C09152=1181.031,74.990,-49.573,-179.182,6.039,148.840
C09153=1181.026,75.239,-49.589,-179.180,6.040,148.840
C09154=1181.021,75.489,-49.607,-179.177,6.041,148.839
C09155=1181.017,75.738,-49.624,-179.175,6.042,148.839
C09156=1181.011,75.987,-49.641,-179.171,6.043,148.838
C09157=1181.006,76.236,-49.659,-179.169,6.044,148.838
C09158=1181.001,76.486,-49.676,-179.167,6.045,148.837
C09159=1180.996,76.736,-49.693,-179.164,6.047,148.837
C09160=1180.992,76.985,-49.710,-179.161,6.047,148.836
C09161=1180.987,77.234,-49.727,-179.159,6.049,148.836
C09162=1180.981,77.483,-49.744,-179.156,6.049,148.835
C09163=1180.977,77.732,-49.762,-179.153,6.051,148.835
C09164=1180.972,77.982,-49.779,-179.151,6.052,148.834
C09165=1180.966,78.232,-49.796,-179.149,6.052,148.834
C09166=1180.962,78.481,-49.814,-179.145,6.054,148.833
C09167=1180.957,78.731,-49.831,-179.143,6.055,148.832
C09168=1180.952,78.980,-49.849,-179.140,6.056,148.832
C09169=1180.948,79.229,-49.866,-179.138,6.057,148.831
C09170=1180.942,79.478,-49.882,-179.135,6.057,148.831
C09171=1180.937,79.727,-49.900,-179.132,6.059,148.830
C09172=1180.932,79.977,-49.917,-179.130,6.060,148.830
C09173=1180.927,80.245,-49.937,-179.127,6.061,148.829
C09174=1180.922,80.514,-49.955,-179.124,6.063,148.829
C09175=1180.916,80.782,-49.974,-179.121,6.063,148.828
C09176=1180.912,81.050,-49.992,-179.119,6.065,148.828
C09177=1180.906,81.300,-50.010,-179.116,6.066,148.827
C09178=1180.901,81.549,-50.028,-179.113,6.067,148.826
C09179=1180.896,81.799,-50.045,-179.111,6.068,148.826
C09180=1180.892,82.048,-50.062,-179.108,6.070,148.825
C09181=1180.887,82.298,-50.080,-179.105,6.070,148.825
C09182=1180.882,82.547,-50.097,-179.103,6.071,148.824
C09183=1180.877,82.796,-50.114,-179.100,6.072,148.824
C09184=1180.873,83.045,-50.132,-179.098,6.073,148.823
C09185=1180.868,83.295,-50.150,-179.095,6.075,148.823
C09186=1180.862,83.544,-50.167,-179.092,6.075,148.822
C09187=1180.858,83.794,-50.185,-179.090,6.077,148.822
C09188=1180.853,84.043,-50.202,-179.087,6.078,148.821
C09189=1180.848,84.292,-50.220,-179.084,6.079,148.821
C09190=1180.843,84.541,-50.238,-179.082,6.080,148.820
C09191=1180.837,84.790,-50.255,-179.079,6.082,148.820
C09192=1180.832,85.040,-50.273,-179.076,6.082,148.819
C09193=1180.828,85.289,-50.290,-179.074,6.083,148.818
C09194=1180.823,85.538,-50.308,-179.071,6.084,148.818
C09195=1180.818,85.787,-50.325,-179.069,6.085,148.817
C09196=1180.813,86.037,-50.343,-179.066,6.087,148.817
C09197=1180.808,86.286,-50.361,-179.064,6.088,148.816
C09198=1180.804,86.536,-50.379,-179.060,6.089,148.816
C09199=1180.800,86.785,-50.396,-179.058,6.090,148.815
C09200=1180.794,87.035,-50.414,-179.055,6.092,148.815
C09201=1180.789,87.284,-50.432,-179.053,6.092,148.814
C09202=1180.785,87.533,-50.450,-179.050,6.094,148.814
C09203=1180.780,87.783,-50.468,-179.048,6.094,148.813
C09204=1180.774,88.032,-50.485,-179.045,6.096,148.813
C09205=1180.769,88.282,-50.503,-179.042,6.097,148.812
C09206=1180.765,88.531,-50.521,-179.039,6.098,148.812
C09207=1180.760,88.780,-50.539,-179.037,6.099,148.811
C09208=1180.755,89.029,-50.557,-179.034,6.101,148.811
C09209=1180.750,89.279,-50.574,-179.031,6.101,148.810
C09210=1180.745,89.528,-50.592,-179.029,6.103,148.810
C09211=1180.740,89.777,-50.609,-179.027,6.104,148.809
C09212=1180.736,90.026,-50.627,-179.023,6.105,148.808
C09213=1180.731,90.275,-50.645,-179.021,6.106,148.808
C09214=1180.726,90.524,-50.663,-179.018,6.107,148.807
C09215=1180.720,90.774,-50.681,-179.016,6.108,148.807
C09216=1180.716,91.024,-50.699,-179.013,6.110,148.806
C09217=1180.711,91.273,-50.717,-179.011,6.111,148.806
C09218=1180.706,91.522,-50.735,-179.008,6.112,148.805
C09219=1180.701,91.772,-50.753,-179.005,6.113,148.805
C09220=1180.697,92.021,-50.771,-179.003,6.115,148.804
C09221=1180.692,92.270,-50.789,-179.000,6.115,148.804
C09222=1180.687,92.519,-50.807,-178.997,6.117,148.803
C09223=1180.682,92.768,-50.825,-178.995,6.117,148.803
C09224=1180.677,93.017,-50.843,-178.992,6.119,148.802
C09225=1180.673,93.267,-50.861,-178.990,6.120,148.802
C09226=1180.668,93.517,-50.879,-178.987,6.121,148.801
C09227=1180.663,93.766,-50.897,-178.984,6.122,148.801
C09228=1180.658,94.015,-50.915,-178.981,6.124,148.800
C09229=1180.652,94.264,-50.934,-178.979,6.125,148.800
C09230=1180.647,94.514,-50.952,-178.976,6.126,148.799
C09231=1180.642,94.763,-50.970,-178.974,6.127,148.799
C09232=1180.638,95.013,-50.988,-178.971,6.129,148.798
C09233=1180.633,95.262,-51.006,-178.968,6.129,148.798
C09234=1180.628,95.511,-51.024,-178.966,6.131,148.797
C09235=1180.623,95.760,-51.042,-178.963,6.131,148.797
C09236=1180.618,96.009,-51.060,-178.960,6.133,148.796
C09237=1180.613,96.258,-51.078,-178.958,6.134,148.795
C09238=1180.609,96.508,-51.096,-178.955,6.135,148.795
C09239=1180.604,96.758,-51.115,-178.952,6.137,148.795
C09240=1180.599,97.007,-51.133,-178.950,6.138,148.794
C09241=1180.594,97.256,-51.151,-178.947,6.139,148.794
C09242=1180.589,97.505,-51.169,-178.944,6.140,148.793
C09243=1180.585,97.755,-51.188,-178.942,6.142,148.793
C09244=1180.580,98.004,-51.206,-178.939,6.143,148.792
C09245=1180.574,98.253,-51.224,-178.936,6.144,148.791
C09246=1180.569,98.502,-51.242,-178.934,6.145,148.791
C09247=1180.565,98.752,-51.261,-178.931,6.146,148.790
C09248=1180.560,99.002,-51.279,-178.929,6.147,148.790
C09249=1180.555,99.250,-51.297,-178.926,6.149,148.790
C09250=1180.551,99.499,-51.315,-178.923,6.150,148.789
C09251=1180.545,99.749,-51.334,-178.921,6.151,148.789
C09252=1180.541,99.999,-51.352,-178.918,6.152,148.788
C09253=1180.536,100.247,-51.371,-178.915,6.153,148.787
C09254=1180.531,100.496,-51.389,-178.913,6.155,148.787
C09255=1180.526,100.747,-51.408,-178.910,6.156,148.786
C09256=1180.521,100.996,-51.426,-178.907,6.157,148.786
C09257=1180.517,101.244,-51.445,-178.905,6.158,148.786
C09258=1180.512,101.493,-51.463,-178.902,6.160,148.785
C09259=1180.507,101.744,-51.482,-178.899,6.161,148.785
C09260=1180.502,101.992,-51.500,-178.897,6.162,148.784
C09261=1180.497,102.241,-51.518,-178.894,6.164,148.784
C09262=1180.492,102.491,-51.536,-178.892,6.165,148.783
C09263=1180.487,102.740,-51.556,-178.889,6.166,148.782
C09264=1180.482,102.989,-51.574,-178.887,6.167,148.782
C09265=1180.478,103.238,-51.592,-178.883,6.168,148.781
C09266=1180.473,103.488,-51.611,-178.881,6.170,148.781
C09267=1180.468,103.737,-51.629,-178.879,6.171,148.781
C09268=1180.463,103.986,-51.647,-178.875,6.172,148.780
C09269=1180.458,104.236,-51.667,-178.873,6.173,148.780
C09270=1180.453,104.485,-51.685,-178.870,6.175,148.779
C09271=1180.449,104.734,-51.704,-178.867,6.176,148.778
C09272=1180.444,104.984,-51.723,-178.865,6.177,148.778
C09273=1180.439,105.233,-51.741,-178.862,6.179,148.778
C09274=1180.433,105.482,-51.760,-178.860,6.179,148.777
C09275=1180.429,105.732,-51.778,-178.857,6.181,148.777
C09276=1180.425,105.980,-51.797,-178.854,6.183,148.776
C09277=1180.419,106.249,-51.817,-178.852,6.183,148.776
C09278=1180.415,106.517,-51.837,-178.849,6.185,148.775
C09279=1180.409,106.786,-51.858,-178.846,6.187,148.775
C09280=1180.403,107.054,-51.878,-178.843,6.188,148.774
C09281=1180.399,107.304,-51.897,-178.841,6.189,148.773
C09282=1180.394,107.553,-51.915,-178.838,6.191,148.773
C09283=1180.389,107.802,-51.934,-178.835,6.192,148.772
C09284=1180.385,108.051,-51.953,-178.833,6.193,148.772
C09285=1180.379,108.300,-51.971,-178.830,6.195,148.772
C09286=1180.375,108.550,-51.991,-178.827,6.195,148.771
C09287=1180.369,108.799,-52.009,-178.824,6.197,148.771
C09288=1180.365,109.048,-52.028,-178.821,6.198,148.770
C09289=1180.360,109.298,-52.047,-178.819,6.199,148.770
C09290=1180.355,109.546,-52.065,-178.816,6.201,148.769
C09291=1180.350,109.796,-52.085,-178.814,6.202,148.768
C09292=1180.345,110.045,-52.103,-178.811,6.203,148.768
C09293=1180.341,110.295,-52.123,-178.808,6.205,148.768
C09294=1180.336,110.543,-52.141,-178.806,6.206,148.767
C09295=1180.330,110.793,-52.160,-178.803,6.207,148.767
C09296=1180.326,111.042,-52.179,-178.800,6.209,148.766
C09297=1180.321,111.291,-52.198,-178.798,6.210,148.766
C09298=1180.317,111.541,-52.217,-178.795,6.211,148.765
C09299=1180.311,111.790,-52.236,-178.792,6.213,148.765
C09300=1180.307,112.039,-52.255,-178.790,6.214,148.764
C09301=1180.302,112.288,-52.274,-178.787,6.215,148.764
C09302=1180.298,112.538,-52.293,-178.785,6.216,148.763
C09303=1180.292,112.787,-52.312,-178.782,6.218,148.763
C09304=1180.288,113.036,-52.332,-178.779,6.219,148.762
C09305=1180.283,113.285,-52.350,-178.777,6.220,148.762
C09306=1180.278,113.535,-52.369,-178.774,6.222,148.761
C09307=1180.273,113.783,-52.388,-178.771,6.223,148.761
C09308=1180.269,114.033,-52.408,-178.769,6.224,148.760
C09309=1180.263,114.282,-52.427,-178.766,6.226,148.760
C09310=1180.259,114.532,-52.445,-178.763,6.227,148.759
C09311=1180.254,114.781,-52.465,-178.761,6.228,148.759
C09312=1180.249,115.030,-52.484,-178.758,6.230,148.759
C09313=1180.244,115.279,-52.503,-178.755,6.231,148.758
C09314=1180.240,115.528,-52.523,-178.753,6.232,148.758
C09315=1180.234,115.777,-52.542,-178.750,6.234,148.757
C09316=1180.230,116.026,-52.561,-178.747,6.235,148.757
C09317=1180.225,116.276,-52.579,-178.745,6.236,148.756
C09318=1180.220,116.525,-52.599,-178.742,6.238,148.756
C09319=1180.215,116.774,-52.618,-178.739,6.240,148.755
C09320=1180.210,117.024,-52.637,-178.737,6.240,148.755
C09321=1180.205,117.272,-52.657,-178.734,6.242,148.754
C09322=1180.201,117.522,-52.676,-178.731,6.244,148.754
C09323=1180.196,117.771,-52.696,-178.729,6.244,148.753
C09324=1180.191,118.020,-52.715,-178.726,6.246,148.753
C09325=1180.186,118.270,-52.734,-178.723,6.248,148.752
C09326=1180.182,118.518,-52.753,-178.721,6.249,148.752
C09327=1180.177,118.768,-52.773,-178.718,6.250,148.751
C09328=1180.172,119.017,-52.792,-178.715,6.252,148.751
C09329=1180.167,119.266,-52.812,-178.713,6.253,148.751
C09330=1180.163,119.516,-52.831,-178.710,6.254,148.750
C09331=1180.157,119.764,-52.850,-178.707,6.256,148.750
C09332=1180.153,120.014,-52.870,-178.705,6.257,148.749
C09333=1180.147,120.263,-52.889,-178.702,6.258,148.749
C09334=1180.143,120.512,-52.908,-178.699,6.260,148.748
C09335=1180.139,120.762,-52.928,-178.697,6.261,148.748
C09336=1180.133,121.011,-52.947,-178.694,6.263,148.747
C09337=1180.129,121.260,-52.967,-178.691,6.264,148.747
C09338=1180.124,121.510,-52.986,-178.689,6.266,148.746
C09339=1180.119,121.758,-53.005,-178.686,6.267,148.746
C09340=1180.115,122.007,-53.025,-178.683,6.268,148.745
C09341=1180.110,122.257,-53.045,-178.681,6.270,148.745
C09342=1180.105,122.506,-53.064,-178.678,6.271,148.744
C09343=1180.100,122.755,-53.084,-178.676,6.273,148.744
C09344=1180.095,123.005,-53.104,-178.673,6.274,148.743
C09345=1180.090,123.254,-53.123,-178.670,6.276,148.743
C09346=1180.086,123.502,-53.143,-178.668,6.277,148.743
C09347=1180.081,123.752,-53.162,-178.665,6.278,148.742
C09348=1180.076,124.001,-53.182,-178.662,6.280,148.742
C09349=1180.071,124.250,-53.201,-178.660,6.281,148.741
C09350=1180.067,124.500,-53.221,-178.657,6.282,148.741
C09351=1180.062,124.748,-53.241,-178.654,6.284,148.740
C09352=1180.057,124.998,-53.261,-178.651,6.286,148.740
C09353=1180.052,125.247,-53.280,-178.649,6.287,148.739
C09354=1180.047,125.496,-53.300,-178.646,6.288,148.739
C09355=1180.042,125.745,-53.320,-178.644,6.290,148.739
C09356=1180.038,125.995,-53.340,-178.641,6.291,148.738
C09357=1180.034,126.244,-53.359,-178.638,6.292,148.738
C09358=1180.028,126.492,-53.379,-178.636,6.294,148.737
C09359=1180.024,126.742,-53.398,-178.633,6.296,148.737
C09360=1180.019,126.991,-53.418,-178.630,6.296,148.736
C09361=1180.014,127.239,-53.438,-178.628,6.298,148.736
C09362=1180.009,127.489,-53.458,-178.625,6.300,148.735
C09363=1180.004,127.739,-53.477,-178.622,6.302,148.735
C09364=1180.000,127.988,-53.498,-178.620,6.302,148.734
C09365=1179.995,128.237,-53.517,-178.617,6.304,148.734
C09366=1179.990,128.486,-53.537,-178.614,6.306,148.734
C09367=1179.986,128.735,-53.557,-178.611,6.307,148.733
C09368=1179.981,128.985,-53.577,-178.609,6.308,148.733
C09369=1179.976,129.233,-53.597,-178.606,6.310,148.732
C09370=1179.971,129.482,-53.616,-178.603,6.311,148.732
C09371=1179.967,129.731,-53.637,-178.601,6.313,148.731
C09372=1179.961,129.981,-53.657,-178.599,6.314,148.731
C09373=1179.956,130.231,-53.677,-178.595,6.316,148.730
C09374=1179.952,130.480,-53.697,-178.593,6.317,148.730
C09375=1179.947,130.729,-53.716,-178.590,6.319,148.730
C09376=1179.942,130.977,-53.737,-178.588,6.320,148.729
C09377=1179.937,131.227,-53.756,-178.585,6.321,148.729
C09378=1179.933,131.476,-53.777,-178.582,6.323,148.728
C09379=1179.928,131.726,-53.796,-178.579,6.325,148.728
C09380=1179.923,131.974,-53.816,-178.577,6.326,148.727
C09381=1179.917,132.243,-53.838,-178.574,6.327,148.727
C09382=1179.913,132.511,-53.860,-178.571,6.329,148.726
C09383=1179.907,132.780,-53.882,-178.569,6.331,148.726
C09384=1179.902,133.048,-53.903,-178.565,6.332,148.725
C09385=1179.898,133.297,-53.923,-178.563,6.334,148.725
C09386=1179.893,133.547,-53.944,-178.560,6.336,148.725
C09387=1179.888,133.796,-53.964,-178.557,6.337,148.724
C09388=1179.884,134.045,-53.984,-178.554,6.339,148.724
C09389=1179.879,134.295,-54.004,-178.552,6.340,148.723
C09390=1179.874,134.544,-54.024,-178.549,6.341,148.723
C09391=1179.869,134.793,-54.045,-178.547,6.343,148.722
C09392=1179.864,135.042,-54.064,-178.544,6.345,148.722
C09393=1179.859,135.291,-54.085,-178.541,6.346,148.721
C09394=1179.855,135.540,-54.105,-178.539,6.347,148.721
C09395=1179.851,135.789,-54.125,-178.536,6.349,148.721
C09396=1179.845,136.039,-54.146,-178.533,6.351,148.720
C09397=1179.841,136.287,-54.166,-178.531,6.352,148.720
C09398=1179.836,136.536,-54.186,-178.528,6.354,148.719
C09399=1179.831,136.786,-54.206,-178.525,6.355,148.719
C09400=1179.826,137.035,-54.227,-178.523,6.357,148.718
C09401=1179.822,137.284,-54.247,-178.520,6.358,148.718
C09402=1179.817,137.532,-54.267,-178.517,6.360,148.718
C09403=1179.812,137.782,-54.287,-178.514,6.362,148.717
C09404=1179.807,138.031,-54.308,-178.512,6.362,148.717
C09405=1179.802,138.280,-54.328,-178.509,6.364,148.716
C09406=1179.798,138.529,-54.349,-178.506,6.366,148.716
C09407=1179.793,138.778,-54.370,-178.504,6.368,148.715
C09408=1179.788,139.027,-54.390,-178.501,6.369,148.715
C09409=1179.784,139.277,-54.410,-178.499,6.370,148.715
C09410=1179.778,139.526,-54.431,-178.496,6.372,148.714
C09411=1179.774,139.775,-54.451,-178.493,6.373,148.714
C09412=1179.770,140.024,-54.471,-178.490,6.375,148.713
C09413=1179.764,140.273,-54.492,-178.488,6.377,148.713
C09414=1179.760,140.522,-54.513,-178.485,6.379,148.712
C09415=1179.756,140.771,-54.533,-178.483,6.380,148.712
C09416=1179.750,141.021,-54.554,-178.480,6.381,148.711
C09417=1179.746,141.269,-54.575,-178.477,6.383,148.711
C09418=1179.740,141.519,-54.595,-178.474,6.385,148.711
C09419=1179.736,141.768,-54.615,-178.472,6.386,148.710
C09420=1179.732,142.017,-54.635,-178.469,6.388,148.710
C09421=1179.726,142.267,-54.656,-178.467,6.389,148.710
C09422=1179.722,142.515,-54.677,-178.464,6.391,148.709
C09423=1179.717,142.765,-54.698,-178.461,6.392,148.709
C09424=1179.712,143.014,-54.718,-178.458,6.394,148.708
C09425=1179.708,143.263,-54.739,-178.456,6.396,148.708
C09426=1179.703,143.512,-54.760,-178.453,6.397,148.707
C09427=1179.698,143.761,-54.780,-178.450,6.399,148.707
C09428=1179.693,144.010,-54.801,-178.448,6.400,148.707
C09429=1179.689,144.258,-54.822,-178.445,6.402,148.706
C09430=1179.684,144.508,-54.843,-178.442,6.403,148.706
C09431=1179.679,144.757,-54.863,-178.440,6.405,148.705
C09432=1179.675,145.007,-54.885,-178.437,6.407,148.705
C09433=1179.670,145.256,-54.905,-178.434,6.409,148.704
C09434=1179.665,145.505,-54.926,-178.431,6.410,148.704
C09435=1179.661,145.754,-54.946,-178.429,6.411,148.704
C09436=1179.656,146.003,-54.967,-178.427,6.413,148.703
C09437=1179.651,146.252,-54.988,-178.424,6.415,148.703
C09438=1179.646,146.501,-55.009,-178.421,6.416,148.702
C09439=1179.642,146.750,-55.030,-178.418,6.418,148.702
C09440=1179.637,146.999,-55.051,-178.415,6.420,148.702
C09441=1179.632,147.248,-55.071,-178.413,6.421,148.701
C09442=1179.627,147.497,-55.092,-178.411,6.422,148.701
C09443=1179.622,147.747,-55.113,-178.408,6.424,148.700
C09444=1179.618,147.995,-55.134,-178.405,6.426,148.700
C09445=1179.613,148.245,-55.155,-178.402,6.428,148.700
C09446=1179.609,148.494,-55.176,-178.399,6.429,148.699
C09447=1179.604,148.743,-55.197,-178.397,6.431,148.699
C09448=1179.599,148.991,-55.218,-178.394,6.433,148.698
C09449=1179.594,149.240,-55.239,-178.391,6.434,148.698
C09450=1179.589,149.490,-55.260,-178.389,6.436,148.698
C09451=1179.585,149.739,-55.281,-178.386,6.437,148.697
C09452=1179.580,149.988,-55.302,-178.384,6.439,148.697
C09453=1179.575,150.237,-55.323,-178.381,6.441,148.696
C09454=1179.571,150.486,-55.344,-178.378,6.442,148.696
C09455=1179.566,150.735,-55.365,-178.376,6.444,148.696
C09456=1179.561,150.984,-55.386,-178.373,6.446,148.695
C09457=1179.557,151.234,-55.407,-178.370,6.447,148.695
C09458=1179.552,151.482,-55.429,-178.367,6.449,148.694
C09459=1179.547,151.732,-55.450,-178.364,6.451,148.694
C09460=1179.543,151.980,-55.471,-178.362,6.453,148.693
C09461=1179.538,152.229,-55.492,-178.360,6.453,148.693
C09462=1179.533,152.479,-55.513,-178.357,6.455,148.693
C09463=1179.528,152.728,-55.535,-178.354,6.457,148.692
C09464=1179.524,152.977,-55.555,-178.352,6.459,148.692
C09465=1179.519,153.225,-55.577,-178.349,6.461,148.692
C09466=1179.514,153.475,-55.598,-178.346,6.462,148.691
C09467=1179.509,153.724,-55.620,-178.344,6.464,148.691
C09468=1179.505,153.973,-55.640,-178.341,6.466,148.690
C09469=1179.500,154.222,-55.662,-178.338,6.467,148.690
C09470=1179.495,154.471,-55.683,-178.335,6.469,148.689
C09471=1179.491,154.720,-55.705,-178.332,6.471,148.689
C09472=1179.486,154.969,-55.725,-178.330,6.473,148.689
C09473=1179.481,155.218,-55.747,-178.327,6.474,148.688
C09474=1179.476,155.467,-55.768,-178.325,6.475,148.688
C09475=1179.472,155.716,-55.790,-178.322,6.477,148.688
C09476=1179.467,155.966,-55.811,-178.319,6.479,148.687
C09477=1179.462,156.214,-55.832,-178.317,6.480,148.687
C09478=1179.457,156.463,-55.853,-178.314,6.482,148.686
C09479=1179.453,156.713,-55.875,-178.311,6.484,148.686
C09480=1179.448,156.961,-55.897,-178.309,6.486,148.686
C09481=1179.443,157.210,-55.918,-178.306,6.488,148.685
C09482=1179.439,157.460,-55.940,-178.303,6.489,148.685
C09483=1179.434,157.708,-55.961,-178.301,6.491,148.685
C09484=1179.429,157.958,-55.982,-178.298,6.493,148.684
C09485=1179.424,158.227,-56.005,-178.295,6.494,148.684
C09486=1179.420,158.495,-56.028,-178.292,6.496,148.683
C09487=1179.414,158.764,-56.052,-178.289,6.498,148.683
C09488=1179.409,159.034,-56.075,-178.286,6.500,148.683
C09489=1179.404,159.282,-56.096,-178.283,6.502,148.682
C09490=1179.400,159.532,-56.118,-178.281,6.504,148.682
C09491=1179.395,159.781,-56.139,-178.278,6.506,148.681
C09492=1179.390,160.029,-56.161,-178.276,6.507,148.681
C09493=1179.386,160.279,-56.183,-178.273,6.508,148.681
C09494=1179.381,160.527,-56.205,-178.271,6.510,148.680
C09495=1179.376,160.776,-56.226,-178.268,6.512,148.680
C09496=1179.372,161.026,-56.248,-178.265,6.514,148.680
C09497=1179.367,161.275,-56.269,-178.263,6.515,148.679
C09498=1179.362,161.523,-56.291,-178.260,6.517,148.679
C09499=1179.358,161.773,-56.313,-178.257,6.519,148.678
C09500=1179.353,162.021,-56.335,-178.254,6.520,148.678
C09501=1179.348,162.271,-56.356,-178.251,6.522,148.677
C09502=1179.343,162.520,-56.378,-178.249,6.524,148.677
C09503=1179.338,162.769,-56.400,-178.246,6.526,148.677
C09504=1179.334,163.018,-56.422,-178.243,6.527,148.676
C09505=1179.329,163.266,-56.443,-178.241,6.529,148.676
C09506=1179.325,163.516,-56.465,-178.238,6.531,148.676
C09507=1179.320,163.764,-56.487,-178.235,6.533,148.675
C09508=1179.316,164.014,-56.509,-178.233,6.535,148.675
C09509=1179.311,164.262,-56.531,-178.230,6.536,148.674
C09510=1179.306,164.512,-56.552,-178.227,6.538,148.674
C09511=1179.302,164.761,-56.574,-178.224,6.540,148.674
C09512=1179.297,165.010,-56.595,-178.222,6.542,148.673
C09513=1179.292,165.259,-56.617,-178.219,6.543,148.673
C09514=1179.287,165.508,-56.640,-178.216,6.545,148.673
C09515=1179.282,165.757,-56.662,-178.214,6.547,148.672
C09516=1179.278,166.006,-56.683,-178.211,6.549,148.672
C09517=1179.273,166.255,-56.706,-178.208,6.550,148.671
C09518=1179.268,166.504,-56.727,-178.206,6.552,148.671
C09519=1179.264,166.753,-56.749,-178.203,6.554,148.671
C09520=1179.260,167.001,-56.772,-178.201,6.556,148.671
C09521=1179.255,167.250,-56.793,-178.198,6.558,148.670
C09522=1179.250,167.500,-56.816,-178.195,6.560,148.670
C09523=1179.245,167.748,-56.838,-178.193,6.561,148.670
C09524=1179.241,167.998,-56.860,-178.190,6.563,148.669
C09525=1179.236,168.246,-56.881,-178.187,6.565,148.669
C09526=1179.232,168.496,-56.903,-178.185,6.567,148.668
C09527=1179.226,168.745,-56.926,-178.182,6.568,148.668
C09528=1179.222,168.994,-56.948,-178.179,6.570,148.668
C09529=1179.217,169.242,-56.969,-178.177,6.572,148.667
C09530=1179.213,169.491,-56.992,-178.174,6.574,148.667
C09531=1179.209,169.741,-57.014,-178.171,6.576,148.667
C09532=1179.203,169.990,-57.037,-178.169,6.577,148.666
C09533=1179.199,170.239,-57.059,-178.166,6.579,148.666
C09534=1179.194,170.487,-57.080,-178.163,6.582,148.665
C09535=1179.190,170.736,-57.103,-178.160,6.583,148.665
C09536=1179.184,170.985,-57.125,-178.157,6.585,148.665
C09537=1179.180,171.235,-57.147,-178.155,6.587,148.664
C09538=1179.175,171.483,-57.169,-178.152,6.589,148.664
C09539=1179.170,171.732,-57.192,-178.149,6.591,148.664
C09540=1179.166,171.981,-57.214,-178.147,6.592,148.663
C09541=1179.161,172.230,-57.236,-178.144,6.594,148.663
C09542=1179.157,172.480,-57.258,-178.141,6.596,148.663
C09543=1179.152,172.728,-57.281,-178.139,6.598,148.662
C09544=1179.147,172.977,-57.303,-178.136,6.599,148.662
C09545=1179.143,173.226,-57.325,-178.134,6.602,148.662
C09546=1179.138,173.475,-57.348,-178.131,6.603,148.661
C09547=1179.134,173.724,-57.370,-178.128,6.605,148.661
C09548=1179.129,173.973,-57.392,-178.126,6.607,148.661
C09549=1179.124,174.222,-57.415,-178.123,6.609,148.660
C09550=1179.119,174.470,-57.437,-178.120,6.610,148.660
C09551=1179.114,174.720,-57.460,-178.118,6.612,148.660
C09552=1179.110,174.969,-57.482,-178.115,6.614,148.659
C09553=1179.105,175.218,-57.504,-178.112,6.617,148.659
C09554=1179.101,175.467,-57.527,-178.109,6.618,148.658
C09555=1179.096,175.716,-57.550,-178.106,6.620,148.658
C09556=1179.091,175.964,-57.573,-178.104,6.622,148.658
C09557=1179.087,176.214,-57.595,-178.101,6.624,148.657
C09558=1179.083,176.462,-57.617,-178.099,6.626,148.657
C09559=1179.077,176.711,-57.640,-178.096,6.628,148.657
C09560=1179.073,176.960,-57.662,-178.093,6.629,148.656
C09561=1179.068,177.210,-57.685,-178.091,6.631,148.656
C09562=1179.064,177.458,-57.707,-178.088,6.633,148.656
C09563=1179.059,177.707,-57.730,-178.085,6.635,148.655
C09564=1179.055,177.956,-57.753,-178.083,6.636,148.655
C09565=1179.049,178.205,-57.775,-178.080,6.638,148.655
C09566=1179.045,178.454,-57.798,-178.077,6.641,148.654
C09567=1179.040,178.703,-57.821,-178.074,6.643,148.654
C09568=1179.036,178.951,-57.843,-178.071,6.644,148.654
C09569=1179.031,179.200,-57.866,-178.069,6.646,148.653
C09570=1179.027,179.450,-57.888,-178.067,6.648,148.653
C09571=1179.022,179.699,-57.912,-178.064,6.650,148.653
C09572=1179.017,179.947,-57.934,-178.061,6.652,148.652
C09573=1179.012,180.196,-57.957,-178.059,6.654,148.652
C09574=1179.008,180.445,-57.979,-178.056,6.655,148.652
C09575=1179.003,180.695,-58.002,-178.053,6.657,148.651
C09576=1178.999,180.943,-58.025,-178.050,6.660,148.651
C09577=1178.994,181.192,-58.048,-178.047,6.662,148.651
C09578=1178.989,181.441,-58.071,-178.045,6.664,148.651
C09579=1178.985,181.690,-58.093,-178.042,6.665,148.650
C09580=1178.980,181.939,-58.116,-178.040,6.667,148.650
C09581=1178.976,182.187,-58.139,-178.037,6.669,148.649
C09582=1178.971,182.437,-58.162,-178.034,6.671,148.649
C09583=1178.966,182.686,-58.185,-178.032,6.673,148.649
C09584=1178.962,182.935,-58.208,-178.028,6.675,148.648
C09585=1178.957,183.183,-58.231,-178.026,6.677,148.648
C09586=1178.953,183.432,-58.254,-178.024,6.679,148.648
C09587=1178.948,183.681,-58.276,-178.021,6.681,148.648
C09588=1178.943,183.930,-58.300,-178.018,6.683,148.647
C09589=1178.939,184.200,-58.324,-178.016,6.684,148.647
C09590=1178.933,184.470,-58.349,-178.012,6.687,148.646
C09591=1178.928,184.739,-58.375,-178.010,6.689,148.646
C09592=1178.924,185.008,-58.399,-178.006,6.691,148.646
C09593=1178.919,185.257,-58.423,-178.004,6.693,148.645
C09594=1178.913,185.506,-58.445,-178.001,6.695,148.645
C09595=1178.909,185.755,-58.468,-177.998,6.697,148.645
C09596=1178.905,186.004,-58.491,-177.996,6.698,148.644
C09597=1178.900,186.253,-58.514,-177.994,6.701,148.644
C09598=1178.895,186.502,-58.538,-177.990,6.703,148.644
C09599=1178.891,186.751,-58.560,-177.988,6.705,148.644
C09600=1178.887,187.000,-58.584,-177.985,6.707,148.643
C09601=1178.881,187.248,-58.607,-177.982,6.709,148.643
C09602=1178.877,187.497,-58.630,-177.980,6.710,148.642
C09603=1178.873,187.746,-58.653,-177.977,6.712,148.642
C09604=1178.868,187.995,-58.676,-177.975,6.714,148.642
C09605=1178.863,188.244,-58.700,-177.971,6.717,148.642
C09606=1178.859,188.493,-58.723,-177.969,6.719,148.641
C09607=1178.855,188.742,-58.746,-177.966,6.720,148.641
C09608=1178.850,188.991,-58.769,-177.964,6.723,148.641
C09609=1178.845,189.239,-58.792,-177.961,6.724,148.640
C09610=1178.840,189.488,-58.816,-177.959,6.726,148.640
C09611=1178.835,189.737,-58.839,-177.955,6.729,148.640
C09612=1178.831,189.986,-58.862,-177.953,6.730,148.639
C09613=1178.826,190.235,-58.886,-177.950,6.732,148.639
C09614=1178.822,190.483,-58.909,-177.948,6.734,148.639
C09615=1178.818,190.732,-58.932,-177.945,6.736,148.639
C09616=1178.813,190.981,-58.956,-177.942,6.738,148.638
C09617=1178.808,191.230,-58.979,-177.939,6.741,148.638
C09618=1178.803,191.479,-59.003,-177.937,6.742,148.638
C09619=1178.799,191.728,-59.026,-177.934,6.744,148.637
C09620=1178.794,191.977,-59.049,-177.932,6.746,148.637
C09621=1178.790,192.226,-59.073,-177.929,6.748,148.637
C09622=1178.785,192.475,-59.097,-177.926,6.751,148.636
C09623=1178.780,192.724,-59.120,-177.923,6.752,148.636
C09624=1178.776,192.973,-59.143,-177.921,6.755,148.636
C09625=1178.772,193.221,-59.167,-177.918,6.756,148.636
C09626=1178.767,193.470,-59.190,-177.916,6.758,148.635
C09627=1178.762,193.719,-59.214,-177.912,6.761,148.635
C09628=1178.758,193.968,-59.237,-177.910,6.763,148.635
C09629=1178.753,194.217,-59.261,-177.907,6.765,148.634
C09630=1178.749,194.466,-59.284,-177.905,6.766,148.634
C09631=1178.744,194.715,-59.308,-177.902,6.768,148.634
C09632=1178.740,194.963,-59.332,-177.899,6.771,148.633
C09633=1178.735,195.212,-59.355,-177.897,6.773,148.633
C09634=1178.730,195.461,-59.379,-177.894,6.775,148.633
C09635=1178.726,195.710,-59.403,-177.891,6.777,148.633
C09636=1178.721,195.959,-59.426,-177.889,6.778,148.632
C09637=1178.716,196.208,-59.449,-177.885,6.781,148.632
C09638=1178.712,196.456,-59.473,-177.883,6.783,148.632
C09639=1178.707,196.705,-59.497,-177.881,6.785,148.631
C09640=1178.702,196.954,-59.521,-177.878,6.787,148.631
C09641=1178.697,197.203,-59.545,-177.875,6.789,148.631
C09642=1178.693,197.452,-59.568,-177.872,6.791,148.631
C09643=1178.688,197.700,-59.592,-177.870,6.793,148.630
C09644=1178.684,197.949,-59.616,-177.867,6.795,148.630
C09645=1178.679,198.198,-59.640,-177.864,6.797,148.630
C09646=1178.675,198.447,-59.663,-177.862,6.800,148.629
C09647=1178.670,198.695,-59.687,-177.859,6.801,148.629
C09648=1178.665,198.944,-59.710,-177.856,6.803,148.629
C09649=1178.662,199.193,-59.735,-177.854,6.805,148.628
C09650=1178.656,199.443,-59.759,-177.851,6.808,148.628
C09651=1178.652,199.691,-59.783,-177.848,6.810,148.628
C09652=1178.647,199.939,-59.807,-177.846,6.812,148.628
C09653=1178.643,200.188,-59.830,-177.843,6.813,148.627
C09654=1178.638,200.437,-59.854,-177.840,6.816,148.627
C09655=1178.634,200.686,-59.878,-177.838,6.818,148.627
C09656=1178.629,200.935,-59.902,-177.835,6.820,148.626
C09657=1178.624,201.184,-59.926,-177.833,6.822,148.626
C09658=1178.620,201.433,-59.950,-177.829,6.825,148.626
C09659=1178.616,201.681,-59.974,-177.827,6.826,148.626
C09660=1178.611,201.930,-59.998,-177.824,6.828,148.625
C09661=1178.606,202.179,-60.022,-177.822,6.830,148.625
C09662=1178.601,202.427,-60.046,-177.819,6.833,148.625
C09663=1178.597,202.677,-60.070,-177.816,6.835,148.625
C09664=1178.593,202.926,-60.094,-177.813,6.837,148.624
C09665=1178.589,203.174,-60.118,-177.811,6.839,148.624
C09666=1178.583,203.423,-60.143,-177.808,6.841,148.624
C09667=1178.579,203.672,-60.166,-177.805,6.843,148.623
C09668=1178.574,203.920,-60.190,-177.803,6.845,148.623
C09669=1178.570,204.170,-60.215,-177.800,6.848,148.623
C09670=1178.565,204.418,-60.239,-177.797,6.850,148.623
C09671=1178.561,204.667,-60.263,-177.795,6.852,148.623
C09672=1178.556,204.915,-60.287,-177.792,6.854,148.622
C09673=1178.552,205.165,-60.312,-177.789,6.856,148.622
C09674=1178.547,205.413,-60.336,-177.786,6.858,148.622
C09675=1178.543,205.662,-60.360,-177.784,6.860,148.621
C09676=1178.538,205.911,-60.384,-177.782,6.862,148.621
C09677=1178.533,206.159,-60.408,-177.778,6.864,148.621
C09678=1178.529,206.409,-60.433,-177.776,6.867,148.621
C09679=1178.524,206.657,-60.457,-177.773,6.868,148.620
C09680=1178.520,206.906,-60.481,-177.770,6.871,148.620
C09681=1178.515,207.154,-60.506,-177.768,6.873,148.620
C09682=1178.511,207.403,-60.530,-177.765,6.875,148.619
C09683=1178.507,207.652,-60.555,-177.762,6.878,148.619
C09684=1178.501,207.901,-60.579,-177.760,6.880,148.619
C09685=1178.497,208.150,-60.603,-177.757,6.882,148.619
C09686=1178.492,208.399,-60.628,-177.755,6.883,148.618
C09687=1178.488,208.648,-60.652,-177.752,6.886,148.618
C09688=1178.483,208.896,-60.676,-177.749,6.888,148.618
C09689=1178.479,209.145,-60.701,-177.747,6.890,148.618
C09690=1178.474,209.394,-60.725,-177.744,6.893,148.617
C09691=1178.469,209.642,-60.749,-177.741,6.895,148.617
C09692=1178.465,209.891,-60.774,-177.738,6.896,148.617
C09693=1178.460,210.162,-60.801,-177.735,6.899,148.617
C09694=1178.455,210.432,-60.827,-177.733,6.901,148.616
C09695=1178.450,210.702,-60.854,-177.730,6.904,148.616
C09696=1178.445,210.973,-60.881,-177.727,6.906,148.616
C09697=1178.440,211.222,-60.906,-177.724,6.908,148.615
C09698=1178.436,211.470,-60.930,-177.722,6.910,148.615
C09699=1178.431,211.720,-60.955,-177.719,6.913,148.615
C09700=1178.427,211.968,-60.979,-177.716,6.915,148.615
C09701=1178.422,212.217,-61.004,-177.714,6.917,148.615
C09702=1178.418,212.465,-61.029,-177.710,6.919,148.614
C09703=1178.413,212.714,-61.053,-177.708,6.921,148.614
C09704=1178.410,212.963,-61.078,-177.706,6.923,148.614
C09705=1178.404,213.212,-61.103,-177.702,6.926,148.613
C09706=1178.400,213.460,-61.127,-177.700,6.928,148.613
C09707=1178.395,213.710,-61.152,-177.698,6.930,148.613
C09708=1178.391,213.958,-61.177,-177.694,6.933,148.613
C09709=1178.386,214.206,-61.201,-177.692,6.935,148.613
C09710=1178.382,214.456,-61.226,-177.689,6.937,148.612
C09711=1178.377,214.704,-61.250,-177.686,6.939,148.612
C09712=1178.373,214.953,-61.276,-177.684,6.941,148.612
C09713=1178.368,215.201,-61.301,-177.681,6.943,148.611
C09714=1178.364,215.450,-61.325,-177.679,6.946,148.611
C09715=1178.359,215.699,-61.351,-177.676,6.948,148.611
C09716=1178.354,215.947,-61.375,-177.673,6.950,148.611
C09717=1178.350,216.196,-61.400,-177.671,6.953,148.611
C09718=1178.346,216.445,-61.425,-177.668,6.954,148.610
C09719=1178.341,216.694,-61.450,-177.665,6.957,148.610
C09720=1178.337,216.942,-61.474,-177.662,6.959,148.610
C09721=1178.332,217.191,-61.500,-177.660,6.961,148.610
C09722=1178.327,217.440,-61.525,-177.657,6.964,148.609
C09723=1178.323,217.689,-61.550,-177.654,6.966,148.609
C09724=1178.319,217.937,-61.574,-177.652,6.967,148.609
C09725=1178.314,218.186,-61.599,-177.649,6.970,148.609
C09726=1178.309,218.435,-61.625,-177.646,6.972,148.608
C09727=1178.305,218.683,-61.649,-177.644,6.974,148.608
C09728=1178.301,218.932,-61.675,-177.641,6.977,148.608
C09729=1178.296,219.181,-61.699,-177.639,6.979,148.608
C09730=1178.291,219.429,-61.725,-177.636,6.982,148.608
C09731=1178.287,219.678,-61.749,-177.633,6.984,148.607
C09732=1178.283,219.927,-61.775,-177.631,6.986,148.607
C09733=1178.278,220.175,-61.800,-177.627,6.988,148.607
C09734=1178.273,220.424,-61.825,-177.625,6.990,148.607
C09735=1178.268,220.673,-61.850,-177.622,6.993,148.606
C09736=1178.265,220.921,-61.875,-177.619,6.995,148.606
C09737=1178.260,221.171,-61.900,-177.617,6.997,148.606
C09738=1178.255,221.419,-61.926,-177.614,7.000,148.606
C09739=1178.251,221.668,-61.951,-177.612,7.002,148.605
C09740=1178.246,221.916,-61.976,-177.609,7.004,148.605
C09741=1178.242,222.165,-62.002,-177.606,7.007,148.605
C09742=1178.237,222.414,-62.026,-177.604,7.008,148.605
C09743=1178.233,222.662,-62.052,-177.601,7.011,148.605
C09744=1178.228,222.911,-62.077,-177.598,7.013,148.604
C09745=1178.224,223.160,-62.102,-177.596,7.015,148.604
C09746=1178.220,223.409,-62.128,-177.593,7.018,148.604
C09747=1178.215,223.657,-62.153,-177.590,7.020,148.604
C09748=1178.210,223.906,-62.178,-177.587,7.023,148.604
C09749=1178.205,224.154,-62.204,-177.585,7.024,148.603
C09750=1178.201,224.403,-62.229,-177.582,7.027,148.603
C09751=1178.197,224.652,-62.255,-177.579,7.029,148.603
C09752=1178.192,224.901,-62.280,-177.577,7.031,148.603
C09753=1178.188,225.150,-62.305,-177.574,7.034,148.602
C09754=1178.183,225.398,-62.331,-177.572,7.036,148.602
C09755=1178.179,225.647,-62.357,-177.569,7.039,148.602
C09756=1178.175,225.896,-62.381,-177.566,7.041,148.602
C09757=1178.170,226.144,-62.406,-177.564,7.043,148.601
C09758=1178.166,226.393,-62.432,-177.561,7.046,148.601
C09759=1178.162,226.641,-62.458,-177.558,7.047,148.601
C09760=1178.157,226.889,-62.483,-177.555,7.050,148.601
C09761=1178.152,227.138,-62.509,-177.553,7.052,148.601
C09762=1178.147,227.387,-62.534,-177.550,7.055,148.600
C09763=1178.142,227.636,-62.560,-177.548,7.057,148.600
C09764=1178.138,227.885,-62.586,-177.545,7.059,148.600
C09765=1178.133,228.133,-62.611,-177.542,7.062,148.600
C09766=1178.129,228.382,-62.637,-177.540,7.064,148.600
C09767=1178.125,228.631,-62.663,-177.537,7.067,148.599
C09768=1178.121,228.879,-62.688,-177.534,7.068,148.599
C09769=1178.116,229.128,-62.714,-177.531,7.071,148.599
C09770=1178.112,229.376,-62.740,-177.529,7.073,148.599
C09771=1178.107,229.625,-62.765,-177.526,7.076,148.599
C09772=1178.103,229.873,-62.791,-177.524,7.078,148.599
C09773=1178.098,230.122,-62.816,-177.521,7.080,148.598
C09774=1178.094,230.371,-62.842,-177.518,7.083,148.598
C09775=1178.089,230.619,-62.868,-177.516,7.085,148.598
C09776=1178.084,230.868,-62.894,-177.513,7.088,148.598
C09777=1178.080,231.117,-62.920,-177.510,7.090,148.597
C09778=1178.076,231.366,-62.945,-177.508,7.092,148.597
C09779=1178.071,231.614,-62.971,-177.505,7.094,148.597
C09780=1178.067,231.863,-62.997,-177.502,7.097,148.597
C09781=1178.062,232.112,-63.023,-177.500,7.099,148.597
C09782=1178.058,232.360,-63.049,-177.497,7.102,148.597
C09783=1178.053,232.609,-63.074,-177.494,7.104,148.596
C09784=1178.049,232.857,-63.101,-177.491,7.107,148.596
C09785=1178.045,233.106,-63.126,-177.489,7.109,148.596
C09786=1178.040,233.355,-63.153,-177.486,7.112,148.596
C09787=1178.035,233.603,-63.178,-177.484,7.114,148.596
C09788=1178.031,233.852,-63.204,-177.481,7.116,148.595
C09789=1178.027,234.100,-63.230,-177.478,7.118,148.595
C09790=1178.022,234.349,-63.257,-177.476,7.120,148.595
C09791=1178.018,234.598,-63.282,-177.473,7.123,148.595
C09792=1178.013,234.846,-63.308,-177.470,7.125,148.595
C09793=1178.008,235.095,-63.333,-177.468,7.128,148.594
C09794=1178.004,235.343,-63.361,-177.465,7.130,148.594
C09795=1178.000,235.592,-63.386,-177.462,7.133,148.594
C09796=1177.995,235.841,-63.412,-177.460,7.135,148.594
C09797=1177.991,236.112,-63.441,-177.457,7.138,148.594
C09798=1177.985,236.384,-63.469,-177.454,7.141,148.594
C09799=1177.981,236.655,-63.498,-177.451,7.143,148.593
C09800=1177.976,236.927,-63.526,-177.448,7.146,148.593
C09801=1177.971,237.175,-63.553,-177.445,7.148,148.593
C09802=1177.967,237.424,-63.579,-177.443,7.151,148.593
C09803=1177.963,237.673,-63.604,-177.440,7.153,148.592
C09804=1177.958,237.921,-63.631,-177.437,7.156,148.592
C09805=1177.953,238.169,-63.657,-177.435,7.158,148.592
C09806=1177.949,238.418,-63.684,-177.432,7.160,148.592
C09807=1177.944,238.667,-63.710,-177.430,7.163,148.592
C09808=1177.940,238.916,-63.735,-177.426,7.165,148.592
C09809=1177.936,239.164,-63.762,-177.424,7.167,148.592
C09810=1177.931,239.413,-63.788,-177.422,7.170,148.591
C09811=1177.927,239.661,-63.815,-177.419,7.172,148.591
C09812=1177.922,239.910,-63.841,-177.416,7.175,148.591
C09813=1177.918,240.159,-63.868,-177.414,7.177,148.591
C09814=1177.913,240.407,-63.893,-177.411,7.180,148.591
C09815=1177.909,240.655,-63.920,-177.409,7.182,148.591
C09816=1177.904,240.904,-63.946,-177.405,7.185,148.590
C09817=1177.900,241.152,-63.973,-177.403,7.188,148.590
C09818=1177.895,241.401,-63.999,-177.400,7.190,148.590
C09819=1177.891,241.649,-64.026,-177.397,7.192,148.590
C09820=1177.887,241.898,-64.053,-177.395,7.195,148.590
C09821=1177.882,242.147,-64.078,-177.392,7.198,148.590
C09822=1177.878,242.395,-64.105,-177.390,7.199,148.589
C09823=1177.873,242.644,-64.131,-177.387,7.202,148.589
C09824=1177.869,242.893,-64.158,-177.384,7.204,148.589
C09825=1177.865,243.141,-64.185,-177.382,7.207,148.589
C09826=1177.860,243.390,-64.211,-177.379,7.209,148.589
C09827=1177.855,243.638,-64.238,-177.376,7.212,148.589
C09828=1177.851,243.887,-64.265,-177.374,7.214,148.588
C09829=1177.846,244.136,-64.291,-177.371,7.217,148.588
C09830=1177.842,244.384,-64.317,-177.368,7.220,148.588
C09831=1177.838,244.632,-64.344,-177.366,7.222,148.588
C09832=1177.834,244.881,-64.371,-177.363,7.225,148.588
C09833=1177.829,245.130,-64.397,-177.360,7.227,148.588
C09834=1177.824,245.378,-64.424,-177.358,7.230,148.588
C09835=1177.820,245.626,-64.451,-177.356,7.232,148.587
C09836=1177.816,245.875,-64.478,-177.353,7.235,148.587
C09837=1177.811,246.124,-64.504,-177.350,7.237,148.587
C09838=1177.807,246.372,-64.531,-177.347,7.239,148.587
C09839=1177.802,246.621,-64.558,-177.345,7.242,148.587
C09840=1177.798,246.869,-64.584,-177.342,7.244,148.587
C09841=1177.794,247.117,-64.611,-177.339,7.247,148.587
C09842=1177.789,247.366,-64.638,-177.337,7.249,148.586
C09843=1177.784,247.615,-64.665,-177.334,7.252,148.586
C09844=1177.780,247.863,-64.691,-177.331,7.255,148.586
C09845=1177.775,248.112,-64.718,-177.329,7.257,148.586
C09846=1177.771,248.360,-64.745,-177.326,7.260,148.586
C09847=1177.767,248.609,-64.772,-177.324,7.262,148.586
C09848=1177.763,248.857,-64.799,-177.321,7.265,148.586
C09849=1177.758,249.106,-64.826,-177.318,7.268,148.585
C09850=1177.753,249.354,-64.853,-177.315,7.270,148.585
C09851=1177.750,249.603,-64.880,-177.313,7.273,148.585
C09852=1177.745,249.851,-64.907,-177.310,7.275,148.585
C09853=1177.740,250.100,-64.934,-177.308,7.278,148.585
C09854=1177.736,250.348,-64.961,-177.305,7.280,148.585
C09855=1177.732,250.596,-64.987,-177.302,7.283,148.585
C09856=1177.727,250.845,-65.014,-177.300,7.285,148.585
C09857=1177.723,251.094,-65.042,-177.297,7.288,148.584
C09858=1177.718,251.343,-65.069,-177.294,7.290,148.584
C09859=1177.714,251.591,-65.096,-177.291,7.293,148.584
C09860=1177.710,251.839,-65.122,-177.289,7.295,148.584
C09861=1177.705,252.088,-65.150,-177.287,7.298,148.584
C09862=1177.700,252.336,-65.177,-177.284,7.300,148.584
C09863=1177.696,252.585,-65.204,-177.281,7.303,148.584
C09864=1177.692,252.833,-65.232,-177.278,7.306,148.584
C09865=1177.687,253.082,-65.259,-177.276,7.308,148.583
C09866=1177.683,253.330,-65.286,-177.273,7.311,148.583
C09867=1177.679,253.578,-65.312,-177.271,7.313,148.583
C09868=1177.674,253.827,-65.339,-177.268,7.316,148.583
C09869=1177.670,254.076,-65.367,-177.265,7.319,148.583
C09870=1177.666,254.324,-65.395,-177.263,7.321,148.583
C09871=1177.661,254.572,-65.422,-177.260,7.324,148.583
C09872=1177.656,254.821,-65.449,-177.257,7.327,148.582
C09873=1177.652,255.069,-65.476,-177.255,7.329,148.582
C09874=1177.648,255.318,-65.504,-177.252,7.332,148.582
C09875=1177.643,255.567,-65.531,-177.250,7.334,148.582
C09876=1177.639,255.815,-65.558,-177.247,7.337,148.582
C09877=1177.634,256.064,-65.585,-177.244,7.340,148.582
C09878=1177.630,256.312,-65.613,-177.242,7.342,148.582
C09879=1177.626,256.561,-65.640,-177.239,7.345,148.582
C09880=1177.621,256.809,-65.667,-177.236,7.347,148.581
C09881=1177.617,257.057,-65.695,-177.234,7.350,148.581
C09882=1177.613,257.306,-65.723,-177.231,7.353,148.581
C09883=1177.608,257.554,-65.750,-177.228,7.356,148.581
C09884=1177.604,257.803,-65.777,-177.226,7.358,148.581
C09885=1177.599,258.051,-65.805,-177.223,7.360,148.581
C09886=1177.595,258.300,-65.833,-177.220,7.363,148.581
C09887=1177.590,258.548,-65.860,-177.218,7.365,148.581
C09888=1177.586,258.796,-65.888,-177.215,7.368,148.581
C09889=1177.581,259.044,-65.915,-177.213,7.371,148.581
C09890=1177.577,259.294,-65.942,-177.211,7.374,148.581
C09891=1177.573,259.542,-65.970,-177.207,7.376,148.580
C09892=1177.568,259.790,-65.997,-177.205,7.379,148.580
C09893=1177.565,260.039,-66.025,-177.202,7.381,148.580
C09894=1177.560,260.287,-66.052,-177.200,7.384,148.580
C09895=1177.556,260.535,-66.080,-177.197,7.387,148.580
C09896=1177.551,260.784,-66.109,-177.195,7.389,148.580
C09897=1177.546,261.032,-66.136,-177.192,7.392,148.580
C09898=1177.542,261.280,-66.163,-177.189,7.395,148.580
C09899=1177.538,261.529,-66.191,-177.187,7.397,148.580
C09900=1177.534,261.777,-66.219,-177.184,7.400,148.579
C09901=1177.529,262.051,-66.249,-177.181,7.403,148.579
C09902=1177.524,262.323,-66.280,-177.178,7.406,148.579
C09903=1177.519,262.597,-66.310,-177.175,7.409,148.579
C09904=1177.514,262.869,-66.341,-177.172,7.412,148.579
C09905=1177.510,263.118,-66.369,-177.170,7.415,148.579
C09906=1177.505,263.366,-66.396,-177.168,7.417,148.579
C09907=1177.502,263.615,-66.424,-177.165,7.420,148.579
C09908=1177.497,263.863,-66.452,-177.162,7.423,148.579
C09909=1177.492,264.112,-66.479,-177.159,7.425,148.579
C09910=1177.488,264.360,-66.508,-177.157,7.428,148.578
C09911=1177.484,264.608,-66.535,-177.154,7.431,148.578
C09912=1177.480,264.857,-66.563,-177.151,7.434,148.578
C09913=1177.475,265.105,-66.591,-177.149,7.436,148.578
C09914=1177.470,265.353,-66.619,-177.146,7.439,148.578
C09915=1177.467,265.602,-66.647,-177.144,7.442,148.578
C09916=1177.462,265.850,-66.675,-177.141,7.444,148.578
C09917=1177.457,266.099,-66.703,-177.139,7.447,148.578
C09918=1177.453,266.347,-66.731,-177.135,7.449,148.578
C09919=1177.449,266.596,-66.759,-177.133,7.452,148.578
C09920=1177.444,266.844,-66.787,-177.131,7.455,148.578
C09921=1177.441,267.092,-66.815,-177.128,7.458,148.578
C09922=1177.435,267.341,-66.844,-177.125,7.460,148.578
C09923=1177.431,267.589,-66.871,-177.123,7.463,148.577
C09924=1177.427,267.838,-66.899,-177.120,7.466,148.577
C09925=1177.422,268.086,-66.927,-177.117,7.469,148.577
C09926=1177.418,268.335,-66.955,-177.115,7.472,148.577
C09927=1177.414,268.582,-66.983,-177.113,7.474,148.577
C09928=1177.409,268.831,-67.012,-177.110,7.477,148.577
C09929=1177.405,269.079,-67.040,-177.107,7.480,148.577
C09930=1177.401,269.328,-67.068,-177.105,7.482,148.577
C09931=1177.396,269.576,-67.096,-177.102,7.484,148.577
C09932=1177.392,269.824,-67.124,-177.099,7.487,148.577
C09933=1177.387,270.073,-67.153,-177.096,7.490,148.577
C09934=1177.384,270.321,-67.181,-177.094,7.493,148.577
C09935=1177.379,270.569,-67.209,-177.091,7.496,148.577
C09936=1177.375,270.818,-67.237,-177.089,7.499,148.577
C09937=1177.370,271.066,-67.266,-177.086,7.502,148.576
C09938=1177.366,271.315,-67.294,-177.084,7.504,148.576
C09939=1177.361,271.564,-67.323,-177.081,7.507,148.576
C09940=1177.357,271.812,-67.350,-177.078,7.510,148.576
C09941=1177.353,272.060,-67.380,-177.075,7.513,148.576
C09942=1177.349,272.308,-67.408,-177.073,7.515,148.576
C09943=1177.344,272.557,-67.436,-177.071,7.518,148.576
C09944=1177.340,272.804,-67.464,-177.068,7.521,148.576
C09945=1177.335,273.053,-67.493,-177.065,7.524,148.576
C09946=1177.331,273.302,-67.521,-177.063,7.526,148.576
C09947=1177.327,273.549,-67.550,-177.060,7.529,148.576
C09948=1177.323,273.798,-67.578,-177.057,7.532,148.576
C09949=1177.318,274.046,-67.607,-177.055,7.535,148.576
C09950=1177.314,274.295,-67.635,-177.053,7.537,148.576
C09951=1177.310,274.544,-67.663,-177.050,7.540,148.576
C09952=1177.305,274.791,-67.693,-177.047,7.543,148.576
C09953=1177.301,275.040,-67.721,-177.044,7.546,148.576
C09954=1177.296,275.288,-67.749,-177.042,7.548,148.576
C09955=1177.293,275.536,-67.778,-177.039,7.551,148.575
C09956=1177.288,275.785,-67.807,-177.037,7.554,148.575
C09957=1177.283,276.033,-67.835,-177.034,7.557,148.575
C09958=1177.280,276.281,-67.864,-177.032,7.559,148.575
C09959=1177.275,276.530,-67.893,-177.029,7.562,148.575
C09960=1177.270,276.778,-67.921,-177.026,7.565,148.575
C09961=1177.267,277.026,-67.950,-177.024,7.568,148.575
C09962=1177.262,277.275,-67.979,-177.021,7.571,148.575
C09963=1177.257,277.523,-68.007,-177.019,7.573,148.575
C09964=1177.253,277.771,-68.036,-177.016,7.576,148.575
C09965=1177.249,278.020,-68.065,-177.013,7.579,148.575
C09966=1177.244,278.268,-68.094,-177.010,7.582,148.575
C09967=1177.240,278.516,-68.122,-177.008,7.584,148.575
C09968=1177.236,278.764,-68.151,-177.006,7.587,148.575
C09969=1177.231,279.013,-68.180,-177.003,7.590,148.575
C09970=1177.228,279.261,-68.208,-177.000,7.593,148.575
C09971=1177.223,279.509,-68.237,-176.997,7.596,148.575
C09972=1177.219,279.758,-68.267,-176.995,7.598,148.575
C09973=1177.214,280.006,-68.295,-176.992,7.601,148.575
C09974=1177.211,280.254,-68.324,-176.990,7.604,148.575
C09975=1177.206,280.503,-68.353,-176.987,7.607,148.575
C09976=1177.202,280.751,-68.382,-176.984,7.610,148.574
C09977=1177.197,280.999,-68.410,-176.982,7.612,148.574
C09978=1177.193,281.247,-68.440,-176.979,7.615,148.574
C09979=1177.189,281.495,-68.469,-176.977,7.618,148.574
C09980=1177.185,281.744,-68.498,-176.974,7.621,148.574
C09981=1177.180,281.992,-68.527,-176.971,7.624,148.574
C09982=1177.175,282.241,-68.555,-176.969,7.627,148.574
C09983=1177.171,282.489,-68.585,-176.967,7.630,148.574
C09984=1177.167,282.737,-68.614,-176.964,7.633,148.574
C09985=1177.162,282.985,-68.643,-176.961,7.636,148.574
C09986=1177.159,283.233,-68.671,-176.958,7.639,148.574
C09987=1177.154,283.482,-68.701,-176.956,7.641,148.574
C09988=1177.150,283.730,-68.730,-176.954,7.644,148.574
C09989=1177.145,283.978,-68.759,-176.951,7.647,148.574
C09990=1177.141,284.226,-68.788,-176.948,7.650,148.574
C09991=1177.137,284.475,-68.818,-176.945,7.653,148.574
C09992=1177.133,284.723,-68.847,-176.943,7.655,148.574
C09993=1177.128,284.972,-68.876,-176.941,7.658,148.574
C09994=1177.124,285.220,-68.905,-176.938,7.661,148.574
C09995=1177.119,285.468,-68.934,-176.935,7.664,148.574
C09996=1177.115,285.716,-68.964,-176.933,7.667,148.574
//INST
///DATE 2021/06/15 17:25
///ATTR SC,RW,RJ
////FRAME ROBOT
///GROUP1 RB1
NOP
MOVL C00000 V=800.0 PL=0
MOVL C00001 V=800.0 PL=0
MOVL C00002 V=800.0 PL=0
MOVL C00003 V=800.0 PL=0
MOVL C00004 V=800.0 PL=0
MOVL C00005 V=800.0 PL=0
MOVL C00006 V=800.0 PL=0
MOVL C00007 V=800.0 PL=0
MOVL C00008 V=800.0 PL=0
MOVL C00009 V=800.0 PL=0
MOVL C00010 V=800.0 PL=0
MOVL C00011 V=800.0 PL=0
MOVL C00012 V=800.0 PL=0
MOVL C00013 V=800.0 PL=0
MOVL C00014 V=800.0 PL=0
MOVL C00015 V=800.0 PL=0
MOVL C00016 V=800.0 PL=0
MOVL C00017 V=800.0 PL=0
MOVL C00018 V=800.0 PL=0
MOVL C00019 V=800.0 PL=0
MOVL C00020 V=800.0 PL=0
MOVL C00021 V=800.0 PL=0
MOVL C00022 V=800.0 PL=0
MOVL C00023 V=800.0 PL=0
MOVL C00024 V=800.0 PL=0
MOVL C00025 V=800.0 PL=0
MOVL C00026 V=800.0 PL=0
MOVL C00027 V=800.0 PL=0
MOVL C00028 V=800.0 PL=0
MOVL C00029 V=800.0 PL=0
MOVL C00030 V=800.0 PL=0
MOVL C00031 V=800.0 PL=0
MOVL C00032 V=800.0 PL=0
MOVL C00033 V=800.0 PL=0
MOVL C00034 V=800.0 PL=0
MOVL C00035 V=800.0 PL=0
MOVL C00036 V=800.0 PL=0
MOVL C00037 V=800.0 PL=0
MOVL C00038 V=800.0 PL=0
MOVL C00039 V=800.0 PL=0
MOVL C00040 V=800.0 PL=0
MOVL C00041 V=800.0 PL=0
MOVL C00042 V=800.0 PL=0
MOVL C00043 V=800.0 PL=0
MOVL C00044 V=800.0 PL=0
MOVL C00045 V=800.0 PL=0
MOVL C00046 V=800.0 PL=0
MOVL C00047 V=800.0 PL=0
MOVL C00048 V=800.0 PL=0
MOVL C00049 V=800.0 PL=0
MOVL C00050 V=800.0 PL=0
MOVL C00051 V=800.0 PL=0
MOVL C00052 V=800.0 PL=0
MOVL C00053 V=800.0 PL=0
MOVL C00054 V=800.0 PL=0
MOVL C00055 V=800.0 PL=0
MOVL C00056 V=800.0 PL=0
MOVL C00057 V=800.0 PL=0
MOVL C00058 V=800.0 PL=0
MOVL C00059 V=800.0 PL=0
MOVL C00060 V=800.0 PL=0
MOVL C00061 V=800.0 PL=0
MOVL C00062 V=800.0 PL=0
MOVL C00063 V=800.0 PL=0
MOVL C00064 V=800.0 PL=0
MOVL C00065 V=800.0 PL=0
MOVL C00066 V=800.0 PL=0
MOVL C00067 V=800.0 PL=0
MOVL C00068 V=800.0 PL=0
MOVL C00069 V=800.0 PL=0
MOVL C00070 V=800.0 PL=0
MOVL C00071 V=800.0 PL=0
MOVL C00072 V=800.0 PL=0
MOVL C00073 V=800.0 PL=0
MOVL C00074 V=800.0 PL=0
MOVL C00075 V=800.0 PL=0
MOVL C00076 V=800.0 PL=0
MOVL C00077 V=800.0 PL=0
MOVL C00078 V=800.0 PL=0
MOVL C00079 V=800.0 PL=0
MOVL C00080 V=800.0 PL=0
MOVL C00081 V=800.0 PL=0
MOVL C00082 V=800.0 PL=0
MOVL C00083 V=800.0 PL=0
MOVL C00084 V=800.0 PL=0
MOVL C00085 V=800.0 PL=0
MOVL C00086 V=800.0 PL=0
MOVL C00087 V=800.0 PL=0
MOVL C00088 V=800.0 PL=0
MOVL C00089 V=800.0 PL=0
MOVL C00090 V=800.0 PL=0
MOVL C00091 V=800.0 PL=0
MOVL C00092 V=800.0 PL=0
MOVL C00093 V=800.0 PL=0
MOVL C00094 V=800.0 PL=0
MOVL C00095 V=800.0 PL=0
MOVL C00096 V=800.0 PL=0
MOVL C00097 V=800.0 PL=0
MOVL C00098 V=800.0 PL=0
MOVL C00099 V=800.0 PL=0
MOVL C00100 V=800.0 PL=0
MOVL C00101 V=800.0 PL=0
MOVL C00102 V=800.0 PL=0
MOVL C00103 V=800.0 PL=0
MOVL C00104 V=800.0 PL=0
MOVL C00105 V=800.0 PL=0
MOVL C00106 V=800.0 PL=0
MOVL C00107 V=800.0 PL=0
MOVL C00108 V=800.0 PL=0
MOVL C00109 V=800.0 PL=0
MOVL C00110 V=800.0 PL=0
MOVL C00111 V=800.0 PL=0
MOVL C00112 V=800.0 PL=0
MOVL C00113 V=800.0 PL=0
MOVL C00114 V=800.0 PL=0
MOVL C00115 V=800.0 PL=0
MOVL C00116 V=800.0 PL=0
MOVL C00117 V=800.0 PL=0
MOVL C00118 V=800.0 PL=0
MOVL C00119 V=800.0 PL=0
MOVL C00120 V=800.0 PL=0
MOVL C00121 V=800.0 PL=0
MOVL C00122 V=800.0 PL=0
MOVL C00123 V=800.0 PL=0
MOVL C00124 V=800.0 PL=0
MOVL C00125 V=800.0 PL=0
MOVL C00126 V=800.0 PL=0
MOVL C00127 V=800.0 PL=0
MOVL C00128 V=800.0 PL=0
MOVL C00129 V=800.0 PL=0
MOVL C00130 V=800.0 PL=0
MOVL C00131 V=800.0 PL=0
MOVL C00132 V=800.0 PL=0
MOVL C00133 V=800.0 PL=0
MOVL C00134 V=800.0 PL=0
MOVL C00135 V=800.0 PL=0
MOVL C00136 V=800.0 PL=0
MOVL C00137 V=800.0 PL=0
MOVL C00138 V=800.0 PL=0
MOVL C00139 V=800.0 PL=0
MOVL C00140 V=800.0 PL=0
MOVL C00141 V=800.0 PL=0
MOVL C00142 V=800.0 PL=0
MOVL C00143 V=800.0 PL=0
MOVL C00144 V=800.0 PL=0
MOVL C00145 V=800.0 PL=0
MOVL C00146 V=800.0 PL=0
MOVL C00147 V=800.0 PL=0
MOVL C00148 V=800.0 PL=0
MOVL C00149 V=800.0 PL=0
MOVL C00150 V=800.0 PL=0
MOVL C00151 V=800.0 PL=0
MOVL C00152 V=800.0 PL=0
MOVL C00153 V=800.0 PL=0
MOVL C00154 V=800.0 PL=0
MOVL C00155 V=800.0 PL=0
MOVL C00156 V=800.0 PL=0
MOVL C00157 V=800.0 PL=0
MOVL C00158 V=800.0 PL=0
MOVL C00159 V=800.0 PL=0
MOVL C00160 V=800.0 PL=0
MOVL C00161 V=800.0 PL=0
MOVL C00162 V=800.0 PL=0
MOVL C00163 V=800.0 PL=0
MOVL C00164 V=800.0 PL=0
MOVL C00165 V=800.0 PL=0
MOVL C00166 V=800.0 PL=0
MOVL C00167 V=800.0 PL=0
MOVL C00168 V=800.0 PL=0
MOVL C00169 V=800.0 PL=0
MOVL C00170 V=800.0 PL=0
MOVL C00171 V=800.0 PL=0
MOVL C00172 V=800.0 PL=0
MOVL C00173 V=800.0 PL=0
MOVL C00174 V=800.0 PL=0
MOVL C00175 V=800.0 PL=0
MOVL C00176 V=800.0 PL=0
MOVL C00177 V=800.0 PL=0
MOVL C00178 V=800.0 PL=0
MOVL C00179 V=800.0 PL=0
MOVL C00180 V=800.0 PL=0
MOVL C00181 V=800.0 PL=0
MOVL C00182 V=800.0 PL=0
MOVL C00183 V=800.0 PL=0
MOVL C00184 V=800.0 PL=0
MOVL C00185 V=800.0 PL=0
MOVL C00186 V=800.0 PL=0
MOVL C00187 V=800.0 PL=0
MOVL C00188 V=800.0 PL=0
MOVL C00189 V=800.0 PL=0
MOVL C00190 V=800.0 PL=0
MOVL C00191 V=800.0 PL=0
MOVL C00192 V=800.0 PL=0
MOVL C00193 V=800.0 PL=0
MOVL C00194 V=800.0 PL=0
MOVL C00195 V=800.0 PL=0
MOVL C00196 V=800.0 PL=0
MOVL C00197 V=800.0 PL=0
MOVL C00198 V=800.0 PL=0
MOVL C00199 V=800.0 PL=0
MOVL C00200 V=800.0 PL=0
MOVL C00201 V=800.0 PL=0
MOVL C00202 V=800.0 PL=0
MOVL C00203 V=800.0 PL=0
MOVL C00204 V=800.0 PL=0
MOVL C00205 V=800.0 PL=0
MOVL C00206 V=800.0 PL=0
MOVL C00207 V=800.0 PL=0
MOVL C00208 V=800.0 PL=0
MOVL C00209 V=800.0 PL=0
MOVL C00210 V=800.0 PL=0
MOVL C00211 V=800.0 PL=0
MOVL C00212 V=800.0 PL=0
MOVL C00213 V=800.0 PL=0
MOVL C00214 V=800.0 PL=0
MOVL C00215 V=800.0 PL=0
MOVL C00216 V=800.0 PL=0
MOVL C00217 V=800.0 PL=0
MOVL C00218 V=800.0 PL=0
MOVL C00219 V=800.0 PL=0
MOVL C00220 V=800.0 PL=0
MOVL C00221 V=800.0 PL=0
MOVL C00222 V=800.0 PL=0
MOVL C00223 V=800.0 PL=0
MOVL C00224 V=800.0 PL=0
MOVL C00225 V=800.0 PL=0
MOVL C00226 V=800.0 PL=0
MOVL C00227 V=800.0 PL=0
MOVL C00228 V=800.0 PL=0
MOVL C00229 V=800.0 PL=0
MOVL C00230 V=800.0 PL=0
MOVL C00231 V=800.0 PL=0
MOVL C00232 V=800.0 PL=0
MOVL C00233 V=800.0 PL=0
MOVL C00234 V=800.0 PL=0
MOVL C00235 V=800.0 PL=0
MOVL C00236 V=800.0 PL=0
MOVL C00237 V=800.0 PL=0
MOVL C00238 V=800.0 PL=0
MOVL C00239 V=800.0 PL=0
MOVL C00240 V=800.0 PL=0
MOVL C00241 V=800.0 PL=0
MOVL C00242 V=800.0 PL=0
MOVL C00243 V=800.0 PL=0
MOVL C00244 V=800.0 PL=0
MOVL C00245 V=800.0 PL=0
MOVL C00246 V=800.0 PL=0
MOVL C00247 V=800.0 PL=0
MOVL C00248 V=800.0 PL=0
MOVL C00249 V=800.0 PL=0
MOVL C00250 V=800.0 PL=0
MOVL C00251 V=800.0 PL=0
MOVL C00252 V=800.0 PL=0
MOVL C00253 V=800.0 PL=0
MOVL C00254 V=800.0 PL=0
MOVL C00255 V=800.0 PL=0
MOVL C00256 V=800.0 PL=0
MOVL C00257 V=800.0 PL=0
MOVL C00258 V=800.0 PL=0
MOVL C00259 V=800.0 PL=0
MOVL C00260 V=800.0 PL=0
MOVL C00261 V=800.0 PL=0
MOVL C00262 V=800.0 PL=0
MOVL C00263 V=800.0 PL=0
MOVL C00264 V=800.0 PL=0
MOVL C00265 V=800.0 PL=0
MOVL C00266 V=800.0 PL=0
MOVL C00267 V=800.0 PL=0
MOVL C00268 V=800.0 PL=0
MOVL C00269 V=800.0 PL=0
MOVL C00270 V=800.0 PL=0
MOVL C00271 V=800.0 PL=0
MOVL C00272 V=800.0 PL=0
MOVL C00273 V=800.0 PL=0
MOVL C00274 V=800.0 PL=0
MOVL C00275 V=800.0 PL=0
MOVL C00276 V=800.0 PL=0
MOVL C00277 V=800.0 PL=0
MOVL C00278 V=800.0 PL=0
MOVL C00279 V=800.0 PL=0
MOVL C00280 V=800.0 PL=0
MOVL C00281 V=800.0 PL=0
MOVL C00282 V=800.0 PL=0
MOVL C00283 V=800.0 PL=0
MOVL C00284 V=800.0 PL=0
MOVL C00285 V=800.0 PL=0
MOVL C00286 V=800.0 PL=0
MOVL C00287 V=800.0 PL=0
MOVL C00288 V=800.0 PL=0
MOVL C00289 V=800.0 PL=0
MOVL C00290 V=800.0 PL=0
MOVL C00291 V=800.0 PL=0
MOVL C00292 V=800.0 PL=0
MOVL C00293 V=800.0 PL=0
MOVL C00294 V=800.0 PL=0
MOVL C00295 V=800.0 PL=0
MOVL C00296 V=800.0 PL=0
MOVL C00297 V=800.0 PL=0
MOVL C00298 V=800.0 PL=0
MOVL C00299 V=800.0 PL=0
MOVL C00300 V=800.0 PL=0
MOVL C00301 V=800.0 PL=0
MOVL C00302 V=800.0 PL=0
MOVL C00303 V=800.0 PL=0
MOVL C00304 V=800.0 PL=0
MOVL C00305 V=800.0 PL=0
MOVL C00306 V=800.0 PL=0
MOVL C00307 V=800.0 PL=0
MOVL C00308 V=800.0 PL=0
MOVL C00309 V=800.0 PL=0
MOVL C00310 V=800.0 PL=0
MOVL C00311 V=800.0 PL=0
MOVL C00312 V=800.0 PL=0
MOVL C00313 V=800.0 PL=0
MOVL C00314 V=800.0 PL=0
MOVL C00315 V=800.0 PL=0
MOVL C00316 V=800.0 PL=0
MOVL C00317 V=800.0 PL=0
MOVL C00318 V=800.0 PL=0
MOVL C00319 V=800.0 PL=0
MOVL C00320 V=800.0 PL=0
MOVL C00321 V=800.0 PL=0
MOVL C00322 V=800.0 PL=0
MOVL C00323 V=800.0 PL=0
MOVL C00324 V=800.0 PL=0
MOVL C00325 V=800.0 PL=0
MOVL C00326 V=800.0 PL=0
MOVL C00327 V=800.0 PL=0
MOVL C00328 V=800.0 PL=0
MOVL C00329 V=800.0 PL=0
MOVL C00330 V=800.0 PL=0
MOVL C00331 V=800.0 PL=0
MOVL C00332 V=800.0 PL=0
MOVL C00333 V=800.0 PL=0
MOVL C00334 V=800.0 PL=0
MOVL C00335 V=800.0 PL=0
MOVL C00336 V=800.0 PL=0
MOVL C00337 V=800.0 PL=0
MOVL C00338 V=800.0 PL=0
MOVL C00339 V=800.0 PL=0
MOVL C00340 V=800.0 PL=0
MOVL C00341 V=800.0 PL=0
MOVL C00342 V=800.0 PL=0
MOVL C00343 V=800.0 PL=0
MOVL C00344 V=800.0 PL=0
MOVL C00345 V=800.0 PL=0
MOVL C00346 V=800.0 PL=0
MOVL C00347 V=800.0 PL=0
MOVL C00348 V=800.0 PL=0
MOVL C00349 V=800.0 PL=0
MOVL C00350 V=800.0 PL=0
MOVL C00351 V=800.0 PL=0
MOVL C00352 V=800.0 PL=0
MOVL C00353 V=800.0 PL=0
MOVL C00354 V=800.0 PL=0
MOVL C00355 V=800.0 PL=0
MOVL C00356 V=800.0 PL=0
MOVL C00357 V=800.0 PL=0
MOVL C00358 V=800.0 PL=0
MOVL C00359 V=800.0 PL=0
MOVL C00360 V=800.0 PL=0
MOVL C00361 V=800.0 PL=0
MOVL C00362 V=800.0 PL=0
MOVL C00363 V=800.0 PL=0
MOVL C00364 V=800.0 PL=0
MOVL C00365 V=800.0 PL=0
MOVL C00366 V=800.0 PL=0
MOVL C00367 V=800.0 PL=0
MOVL C00368 V=800.0 PL=0
MOVL C00369 V=800.0 PL=0
MOVL C00370 V=800.0 PL=0
MOVL C00371 V=800.0 PL=0
MOVL C00372 V=800.0 PL=0
MOVL C00373 V=800.0 PL=0
MOVL C00374 V=800.0 PL=0
MOVL C00375 V=800.0 PL=0
MOVL C00376 V=800.0 PL=0
MOVL C00377 V=800.0 PL=0
MOVL C00378 V=800.0 PL=0
MOVL C00379 V=800.0 PL=0
MOVL C00380 V=800.0 PL=0
MOVL C00381 V=800.0 PL=0
MOVL C00382 V=800.0 PL=0
MOVL C00383 V=800.0 PL=0
MOVL C00384 V=800.0 PL=0
MOVL C00385 V=800.0 PL=0
MOVL C00386 V=800.0 PL=0
MOVL C00387 V=800.0 PL=0
MOVL C00388 V=800.0 PL=0
MOVL C00389 V=800.0 PL=0
MOVL C00390 V=800.0 PL=0
MOVL C00391 V=800.0 PL=0
MOVL C00392 V=800.0 PL=0
MOVL C00393 V=800.0 PL=0
MOVL C00394 V=800.0 PL=0
MOVL C00395 V=800.0 PL=0
MOVL C00396 V=800.0 PL=0
MOVL C00397 V=800.0 PL=0
MOVL C00398 V=800.0 PL=0
MOVL C00399 V=800.0 PL=0
MOVL C00400 V=800.0 PL=0
MOVL C00401 V=800.0 PL=0
MOVL C00402 V=800.0 PL=0
MOVL C00403 V=800.0 PL=0
MOVL C00404 V=800.0 PL=0
MOVL C00405 V=800.0 PL=0
MOVL C00406 V=800.0 PL=0
MOVL C00407 V=800.0 PL=0
MOVL C00408 V=800.0 PL=0
MOVL C00409 V=800.0 PL=0
MOVL C00410 V=800.0 PL=0
MOVL C00411 V=800.0 PL=0
MOVL C00412 V=800.0 PL=0
MOVL C00413 V=800.0 PL=0
MOVL C00414 V=800.0 PL=0
MOVL C00415 V=800.0 PL=0
MOVL C00416 V=800.0 PL=0
MOVL C00417 V=800.0 PL=0
MOVL C00418 V=800.0 PL=0
MOVL C00419 V=800.0 PL=0
MOVL C00420 V=800.0 PL=0
MOVL C00421 V=800.0 PL=0
MOVL C00422 V=800.0 PL=0
MOVL C00423 V=800.0 PL=0
MOVL C00424 V=800.0 PL=0
MOVL C00425 V=800.0 PL=0
MOVL C00426 V=800.0 PL=0
MOVL C00427 V=800.0 PL=0
MOVL C00428 V=800.0 PL=0
MOVL C00429 V=800.0 PL=0
MOVL C00430 V=800.0 PL=0
MOVL C00431 V=800.0 PL=0
MOVL C00432 V=800.0 PL=0
MOVL C00433 V=800.0 PL=0
MOVL C00434 V=800.0 PL=0
MOVL C00435 V=800.0 PL=0
MOVL C00436 V=800.0 PL=0
MOVL C00437 V=800.0 PL=0
MOVL C00438 V=800.0 PL=0
MOVL C00439 V=800.0 PL=0
MOVL C00440 V=800.0 PL=0
MOVL C00441 V=800.0 PL=0
MOVL C00442 V=800.0 PL=0
MOVL C00443 V=800.0 PL=0
MOVL C00444 V=800.0 PL=0
MOVL C00445 V=800.0 PL=0
MOVL C00446 V=800.0 PL=0
MOVL C00447 V=800.0 PL=0
MOVL C00448 V=800.0 PL=0
MOVL C00449 V=800.0 PL=0
MOVL C00450 V=800.0 PL=0
MOVL C00451 V=800.0 PL=0
MOVL C00452 V=800.0 PL=0
MOVL C00453 V=800.0 PL=0
MOVL C00454 V=800.0 PL=0
MOVL C00455 V=800.0 PL=0
MOVL C00456 V=800.0 PL=0
MOVL C00457 V=800.0 PL=0
MOVL C00458 V=800.0 PL=0
MOVL C00459 V=800.0 PL=0
MOVL C00460 V=800.0 PL=0
MOVL C00461 V=800.0 PL=0
MOVL C00462 V=800.0 PL=0
MOVL C00463 V=800.0 PL=0
MOVL C00464 V=800.0 PL=0
MOVL C00465 V=800.0 PL=0
MOVL C00466 V=800.0 PL=0
MOVL C00467 V=800.0 PL=0
MOVL C00468 V=800.0 PL=0
MOVL C00469 V=800.0 PL=0
MOVL C00470 V=800.0 PL=0
MOVL C00471 V=800.0 PL=0
MOVL C00472 V=800.0 PL=0
MOVL C00473 V=800.0 PL=0
MOVL C00474 V=800.0 PL=0
MOVL C00475 V=800.0 PL=0
MOVL C00476 V=800.0 PL=0
MOVL C00477 V=800.0 PL=0
MOVL C00478 V=800.0 PL=0
MOVL C00479 V=800.0 PL=0
MOVL C00480 V=800.0 PL=0
MOVL C00481 V=800.0 PL=0
MOVL C00482 V=800.0 PL=0
MOVL C00483 V=800.0 PL=0
MOVL C00484 V=800.0 PL=0
MOVL C00485 V=800.0 PL=0
MOVL C00486 V=800.0 PL=0
MOVL C00487 V=800.0 PL=0
MOVL C00488 V=800.0 PL=0
MOVL C00489 V=800.0 PL=0
MOVL C00490 V=800.0 PL=0
MOVL C00491 V=800.0 PL=0
MOVL C00492 V=800.0 PL=0
MOVL C00493 V=800.0 PL=0
MOVL C00494 V=800.0 PL=0
MOVL C00495 V=800.0 PL=0
MOVL C00496 V=800.0 PL=0
MOVL C00497 V=800.0 PL=0
MOVL C00498 V=800.0 PL=0
MOVL C00499 V=800.0 PL=0
MOVL C00500 V=800.0 PL=0
MOVL C00501 V=800.0 PL=0
MOVL C00502 V=800.0 PL=0
MOVL C00503 V=800.0 PL=0
MOVL C00504 V=800.0 PL=0
MOVL C00505 V=800.0 PL=0
MOVL C00506 V=800.0 PL=0
MOVL C00507 V=800.0 PL=0
MOVL C00508 V=800.0 PL=0
MOVL C00509 V=800.0 PL=0
MOVL C00510 V=800.0 PL=0
MOVL C00511 V=800.0 PL=0
MOVL C00512 V=800.0 PL=0
MOVL C00513 V=800.0 PL=0
MOVL C00514 V=800.0 PL=0
MOVL C00515 V=800.0 PL=0
MOVL C00516 V=800.0 PL=0
MOVL C00517 V=800.0 PL=0
MOVL C00518 V=800.0 PL=0
MOVL C00519 V=800.0 PL=0
MOVL C00520 V=800.0 PL=0
MOVL C00521 V=800.0 PL=0
MOVL C00522 V=800.0 PL=0
MOVL C00523 V=800.0 PL=0
MOVL C00524 V=800.0 PL=0
MOVL C00525 V=800.0 PL=0
MOVL C00526 V=800.0 PL=0
MOVL C00527 V=800.0 PL=0
MOVL C00528 V=800.0 PL=0
MOVL C00529 V=800.0 PL=0
MOVL C00530 V=800.0 PL=0
MOVL C00531 V=800.0 PL=0
MOVL C00532 V=800.0 PL=0
MOVL C00533 V=800.0 PL=0
MOVL C00534 V=800.0 PL=0
MOVL C00535 V=800.0 PL=0
MOVL C00536 V=800.0 PL=0
MOVL C00537 V=800.0 PL=0
MOVL C00538 V=800.0 PL=0
MOVL C00539 V=800.0 PL=0
MOVL C00540 V=800.0 PL=0
MOVL C00541 V=800.0 PL=0
MOVL C00542 V=800.0 PL=0
MOVL C00543 V=800.0 PL=0
MOVL C00544 V=800.0 PL=0
MOVL C00545 V=800.0 PL=0
MOVL C00546 V=800.0 PL=0
MOVL C00547 V=800.0 PL=0
MOVL C00548 V=800.0 PL=0
MOVL C00549 V=800.0 PL=0
MOVL C00550 V=800.0 PL=0
MOVL C00551 V=800.0 PL=0
MOVL C00552 V=800.0 PL=0
MOVL C00553 V=800.0 PL=0
MOVL C00554 V=800.0 PL=0
MOVL C00555 V=800.0 PL=0
MOVL C00556 V=800.0 PL=0
MOVL C00557 V=800.0 PL=0
MOVL C00558 V=800.0 PL=0
MOVL C00559 V=800.0 PL=0
MOVL C00560 V=800.0 PL=0
MOVL C00561 V=800.0 PL=0
MOVL C00562 V=800.0 PL=0
MOVL C00563 V=800.0 PL=0
MOVL C00564 V=800.0 PL=0
MOVL C00565 V=800.0 PL=0
MOVL C00566 V=800.0 PL=0
MOVL C00567 V=800.0 PL=0
MOVL C00568 V=800.0 PL=0
MOVL C00569 V=800.0 PL=0
MOVL C00570 V=800.0 PL=0
MOVL C00571 V=800.0 PL=0
MOVL C00572 V=800.0 PL=0
MOVL C00573 V=800.0 PL=0
MOVL C00574 V=800.0 PL=0
MOVL C00575 V=800.0 PL=0
MOVL C00576 V=800.0 PL=0
MOVL C00577 V=800.0 PL=0
MOVL C00578 V=800.0 PL=0
MOVL C00579 V=800.0 PL=0
MOVL C00580 V=800.0 PL=0
MOVL C00581 V=800.0 PL=0
MOVL C00582 V=800.0 PL=0
MOVL C00583 V=800.0 PL=0
MOVL C00584 V=800.0 PL=0
MOVL C00585 V=800.0 PL=0
MOVL C00586 V=800.0 PL=0
MOVL C00587 V=800.0 PL=0
MOVL C00588 V=800.0 PL=0
MOVL C00589 V=800.0 PL=0
MOVL C00590 V=800.0 PL=0
MOVL C00591 V=800.0 PL=0
MOVL C00592 V=800.0 PL=0
MOVL C00593 V=800.0 PL=0
MOVL C00594 V=800.0 PL=0
MOVL C00595 V=800.0 PL=0
MOVL C00596 V=800.0 PL=0
MOVL C00597 V=800.0 PL=0
MOVL C00598 V=800.0 PL=0
MOVL C00599 V=800.0 PL=0
MOVL C00600 V=800.0 PL=0
MOVL C00601 V=800.0 PL=0
MOVL C00602 V=800.0 PL=0
MOVL C00603 V=800.0 PL=0
MOVL C00604 V=800.0 PL=0
MOVL C00605 V=800.0 PL=0
MOVL C00606 V=800.0 PL=0
MOVL C00607 V=800.0 PL=0
MOVL C00608 V=800.0 PL=0
MOVL C00609 V=800.0 PL=0
MOVL C00610 V=800.0 PL=0
MOVL C00611 V=800.0 PL=0
MOVL C00612 V=800.0 PL=0
MOVL C00613 V=800.0 PL=0
MOVL C00614 V=800.0 PL=0
MOVL C00615 V=800.0 PL=0
MOVL C00616 V=800.0 PL=0
MOVL C00617 V=800.0 PL=0
MOVL C00618 V=800.0 PL=0
MOVL C00619 V=800.0 PL=0
MOVL C00620 V=800.0 PL=0
MOVL C00621 V=800.0 PL=0
MOVL C00622 V=800.0 PL=0
MOVL C00623 V=800.0 PL=0
MOVL C00624 V=800.0 PL=0
MOVL C00625 V=800.0 PL=0
MOVL C00626 V=800.0 PL=0
MOVL C00627 V=800.0 PL=0
MOVL C00628 V=800.0 PL=0
MOVL C00629 V=800.0 PL=0
MOVL C00630 V=800.0 PL=0
MOVL C00631 V=800.0 PL=0
MOVL C00632 V=800.0 PL=0
MOVL C00633 V=800.0 PL=0
MOVL C00634 V=800.0 PL=0
MOVL C00635 V=800.0 PL=0
MOVL C00636 V=800.0 PL=0
MOVL C00637 V=800.0 PL=0
MOVL C00638 V=800.0 PL=0
MOVL C00639 V=800.0 PL=0
MOVL C00640 V=800.0 PL=0
MOVL C00641 V=800.0 PL=0
MOVL C00642 V=800.0 PL=0
MOVL C00643 V=800.0 PL=0
MOVL C00644 V=800.0 PL=0
MOVL C00645 V=800.0 PL=0
MOVL C00646 V=800.0 PL=0
MOVL C00647 V=800.0 PL=0
MOVL C00648 V=800.0 PL=0
MOVL C00649 V=800.0 PL=0
MOVL C00650 V=800.0 PL=0
MOVL C00651 V=800.0 PL=0
MOVL C00652 V=800.0 PL=0
MOVL C00653 V=800.0 PL=0
MOVL C00654 V=800.0 PL=0
MOVL C00655 V=800.0 PL=0
MOVL C00656 V=800.0 PL=0
MOVL C00657 V=800.0 PL=0
MOVL C00658 V=800.0 PL=0
MOVL C00659 V=800.0 PL=0
MOVL C00660 V=800.0 PL=0
MOVL C00661 V=800.0 PL=0
MOVL C00662 V=800.0 PL=0
MOVL C00663 V=800.0 PL=0
MOVL C00664 V=800.0 PL=0
MOVL C00665 V=800.0 PL=0
MOVL C00666 V=800.0 PL=0
MOVL C00667 V=800.0 PL=0
MOVL C00668 V=800.0 PL=0
MOVL C00669 V=800.0 PL=0
MOVL C00670 V=800.0 PL=0
MOVL C00671 V=800.0 PL=0
MOVL C00672 V=800.0 PL=0
MOVL C00673 V=800.0 PL=0
MOVL C00674 V=800.0 PL=0
MOVL C00675 V=800.0 PL=0
MOVL C00676 V=800.0 PL=0
MOVL C00677 V=800.0 PL=0
MOVL C00678 V=800.0 PL=0
MOVL C00679 V=800.0 PL=0
MOVL C00680 V=800.0 PL=0
MOVL C00681 V=800.0 PL=0
MOVL C00682 V=800.0 PL=0
MOVL C00683 V=800.0 PL=0
MOVL C00684 V=800.0 PL=0
MOVL C00685 V=800.0 PL=0
MOVL C00686 V=800.0 PL=0
MOVL C00687 V=800.0 PL=0
MOVL C00688 V=800.0 PL=0
MOVL C00689 V=800.0 PL=0
MOVL C00690 V=800.0 PL=0
MOVL C00691 V=800.0 PL=0
MOVL C00692 V=800.0 PL=0
MOVL C00693 V=800.0 PL=0
MOVL C00694 V=800.0 PL=0
MOVL C00695 V=800.0 PL=0
MOVL C00696 V=800.0 PL=0
MOVL C00697 V=800.0 PL=0
MOVL C00698 V=800.0 PL=0
MOVL C00699 V=800.0 PL=0
MOVL C00700 V=800.0 PL=0
MOVL C00701 V=800.0 PL=0
MOVL C00702 V=800.0 PL=0
MOVL C00703 V=800.0 PL=0
MOVL C00704 V=800.0 PL=0
MOVL C00705 V=800.0 PL=0
MOVL C00706 V=800.0 PL=0
MOVL C00707 V=800.0 PL=0
MOVL C00708 V=800.0 PL=0
MOVL C00709 V=800.0 PL=0
MOVL C00710 V=800.0 PL=0
MOVL C00711 V=800.0 PL=0
MOVL C00712 V=800.0 PL=0
MOVL C00713 V=800.0 PL=0
MOVL C00714 V=800.0 PL=0
MOVL C00715 V=800.0 PL=0
MOVL C00716 V=800.0 PL=0
MOVL C00717 V=800.0 PL=0
MOVL C00718 V=800.0 PL=0
MOVL C00719 V=800.0 PL=0
MOVL C00720 V=800.0 PL=0
MOVL C00721 V=800.0 PL=0
MOVL C00722 V=800.0 PL=0
MOVL C00723 V=800.0 PL=0
MOVL C00724 V=800.0 PL=0
MOVL C00725 V=800.0 PL=0
MOVL C00726 V=800.0 PL=0
MOVL C00727 V=800.0 PL=0
MOVL C00728 V=800.0 PL=0
MOVL C00729 V=800.0 PL=0
MOVL C00730 V=800.0 PL=0
MOVL C00731 V=800.0 PL=0
MOVL C00732 V=800.0 PL=0
MOVL C00733 V=800.0 PL=0
MOVL C00734 V=800.0 PL=0
MOVL C00735 V=800.0 PL=0
MOVL C00736 V=800.0 PL=0
MOVL C00737 V=800.0 PL=0
MOVL C00738 V=800.0 PL=0
MOVL C00739 V=800.0 PL=0
MOVL C00740 V=800.0 PL=0
MOVL C00741 V=800.0 PL=0
MOVL C00742 V=800.0 PL=0
MOVL C00743 V=800.0 PL=0
MOVL C00744 V=800.0 PL=0
MOVL C00745 V=800.0 PL=0
MOVL C00746 V=800.0 PL=0
MOVL C00747 V=800.0 PL=0
MOVL C00748 V=800.0 PL=0
MOVL C00749 V=800.0 PL=0
MOVL C00750 V=800.0 PL=0
MOVL C00751 V=800.0 PL=0
MOVL C00752 V=800.0 PL=0
MOVL C00753 V=800.0 PL=0
MOVL C00754 V=800.0 PL=0
MOVL C00755 V=800.0 PL=0
MOVL C00756 V=800.0 PL=0
MOVL C00757 V=800.0 PL=0
MOVL C00758 V=800.0 PL=0
MOVL C00759 V=800.0 PL=0
MOVL C00760 V=800.0 PL=0
MOVL C00761 V=800.0 PL=0
MOVL C00762 V=800.0 PL=0
MOVL C00763 V=800.0 PL=0
MOVL C00764 V=800.0 PL=0
MOVL C00765 V=800.0 PL=0
MOVL C00766 V=800.0 PL=0
MOVL C00767 V=800.0 PL=0
MOVL C00768 V=800.0 PL=0
MOVL C00769 V=800.0 PL=0
MOVL C00770 V=800.0 PL=0
MOVL C00771 V=800.0 PL=0
MOVL C00772 V=800.0 PL=0
MOVL C00773 V=800.0 PL=0
MOVL C00774 V=800.0 PL=0
MOVL C00775 V=800.0 PL=0
MOVL C00776 V=800.0 PL=0
MOVL C00777 V=800.0 PL=0
MOVL C00778 V=800.0 PL=0
MOVL C00779 V=800.0 PL=0
MOVL C00780 V=800.0 PL=0
MOVL C00781 V=800.0 PL=0
MOVL C00782 V=800.0 PL=0
MOVL C00783 V=800.0 PL=0
MOVL C00784 V=800.0 PL=0
MOVL C00785 V=800.0 PL=0
MOVL C00786 V=800.0 PL=0
MOVL C00787 V=800.0 PL=0
MOVL C00788 V=800.0 PL=0
MOVL C00789 V=800.0 PL=0
MOVL C00790 V=800.0 PL=0
MOVL C00791 V=800.0 PL=0
MOVL C00792 V=800.0 PL=0
MOVL C00793 V=800.0 PL=0
MOVL C00794 V=800.0 PL=0
MOVL C00795 V=800.0 PL=0
MOVL C00796 V=800.0 PL=0
MOVL C00797 V=800.0 PL=0
MOVL C00798 V=800.0 PL=0
MOVL C00799 V=800.0 PL=0
MOVL C00800 V=800.0 PL=0
MOVL C00801 V=800.0 PL=0
MOVL C00802 V=800.0 PL=0
MOVL C00803 V=800.0 PL=0
MOVL C00804 V=800.0 PL=0
MOVL C00805 V=800.0 PL=0
MOVL C00806 V=800.0 PL=0
MOVL C00807 V=800.0 PL=0
MOVL C00808 V=800.0 PL=0
MOVL C00809 V=800.0 PL=0
MOVL C00810 V=800.0 PL=0
MOVL C00811 V=800.0 PL=0
MOVL C00812 V=800.0 PL=0
MOVL C00813 V=800.0 PL=0
MOVL C00814 V=800.0 PL=0
MOVL C00815 V=800.0 PL=0
MOVL C00816 V=800.0 PL=0
MOVL C00817 V=800.0 PL=0
MOVL C00818 V=800.0 PL=0
MOVL C00819 V=800.0 PL=0
MOVL C00820 V=800.0 PL=0
MOVL C00821 V=800.0 PL=0
MOVL C00822 V=800.0 PL=0
MOVL C00823 V=800.0 PL=0
MOVL C00824 V=800.0 PL=0
MOVL C00825 V=800.0 PL=0
MOVL C00826 V=800.0 PL=0
MOVL C00827 V=800.0 PL=0
MOVL C00828 V=800.0 PL=0
MOVL C00829 V=800.0 PL=0
MOVL C00830 V=800.0 PL=0
MOVL C00831 V=800.0 PL=0
MOVL C00832 V=800.0 PL=0
MOVL C00833 V=800.0 PL=0
MOVL C00834 V=800.0 PL=0
MOVL C00835 V=800.0 PL=0
MOVL C00836 V=800.0 PL=0
MOVL C00837 V=800.0 PL=0
MOVL C00838 V=800.0 PL=0
MOVL C00839 V=800.0 PL=0
MOVL C00840 V=800.0 PL=0
MOVL C00841 V=800.0 PL=0
MOVL C00842 V=800.0 PL=0
MOVL C00843 V=800.0 PL=0
MOVL C00844 V=800.0 PL=0
MOVL C00845 V=800.0 PL=0
MOVL C00846 V=800.0 PL=0
MOVL C00847 V=800.0 PL=0
MOVL C00848 V=800.0 PL=0
MOVL C00849 V=800.0 PL=0
MOVL C00850 V=800.0 PL=0
MOVL C00851 V=800.0 PL=0
MOVL C00852 V=800.0 PL=0
MOVL C00853 V=800.0 PL=0
MOVL C00854 V=800.0 PL=0
MOVL C00855 V=800.0 PL=0
MOVL C00856 V=800.0 PL=0
MOVL C00857 V=800.0 PL=0
MOVL C00858 V=800.0 PL=0
MOVL C00859 V=800.0 PL=0
MOVL C00860 V=800.0 PL=0
MOVL C00861 V=800.0 PL=0
MOVL C00862 V=800.0 PL=0
MOVL C00863 V=800.0 PL=0
MOVL C00864 V=800.0 PL=0
MOVL C00865 V=800.0 PL=0
MOVL C00866 V=800.0 PL=0
MOVL C00867 V=800.0 PL=0
MOVL C00868 V=800.0 PL=0
MOVL C00869 V=800.0 PL=0
MOVL C00870 V=800.0 PL=0
MOVL C00871 V=800.0 PL=0
MOVL C00872 V=800.0 PL=0
MOVL C00873 V=800.0 PL=0
MOVL C00874 V=800.0 PL=0
MOVL C00875 V=800.0 PL=0
MOVL C00876 V=800.0 PL=0
MOVL C00877 V=800.0 PL=0
MOVL C00878 V=800.0 PL=0
MOVL C00879 V=800.0 PL=0
MOVL C00880 V=800.0 PL=0
MOVL C00881 V=800.0 PL=0
MOVL C00882 V=800.0 PL=0
MOVL C00883 V=800.0 PL=0
MOVL C00884 V=800.0 PL=0
MOVL C00885 V=800.0 PL=0
MOVL C00886 V=800.0 PL=0
MOVL C00887 V=800.0 PL=0
MOVL C00888 V=800.0 PL=0
MOVL C00889 V=800.0 PL=0
MOVL C00890 V=800.0 PL=0
MOVL C00891 V=800.0 PL=0
MOVL C00892 V=800.0 PL=0
MOVL C00893 V=800.0 PL=0
MOVL C00894 V=800.0 PL=0
MOVL C00895 V=800.0 PL=0
MOVL C00896 V=800.0 PL=0
MOVL C00897 V=800.0 PL=0
MOVL C00898 V=800.0 PL=0
MOVL C00899 V=800.0 PL=0
MOVL C00900 V=800.0 PL=0
MOVL C00901 V=800.0 PL=0
MOVL C00902 V=800.0 PL=0
MOVL C00903 V=800.0 PL=0
MOVL C00904 V=800.0 PL=0
MOVL C00905 V=800.0 PL=0
MOVL C00906 V=800.0 PL=0
MOVL C00907 V=800.0 PL=0
MOVL C00908 V=800.0 PL=0
MOVL C00909 V=800.0 PL=0
MOVL C00910 V=800.0 PL=0
MOVL C00911 V=800.0 PL=0
MOVL C00912 V=800.0 PL=0
MOVL C00913 V=800.0 PL=0
MOVL C00914 V=800.0 PL=0
MOVL C00915 V=800.0 PL=0
MOVL C00916 V=800.0 PL=0
MOVL C00917 V=800.0 PL=0
MOVL C00918 V=800.0 PL=0
MOVL C00919 V=800.0 PL=0
MOVL C00920 V=800.0 PL=0
MOVL C00921 V=800.0 PL=0
MOVL C00922 V=800.0 PL=0
MOVL C00923 V=800.0 PL=0
MOVL C00924 V=800.0 PL=0
MOVL C00925 V=800.0 PL=0
MOVL C00926 V=800.0 PL=0
MOVL C00927 V=800.0 PL=0
MOVL C00928 V=800.0 PL=0
MOVL C00929 V=800.0 PL=0
MOVL C00930 V=800.0 PL=0
MOVL C00931 V=800.0 PL=0
MOVL C00932 V=800.0 PL=0
MOVL C00933 V=800.0 PL=0
MOVL C00934 V=800.0 PL=0
MOVL C00935 V=800.0 PL=0
MOVL C00936 V=800.0 PL=0
MOVL C00937 V=800.0 PL=0
MOVL C00938 V=800.0 PL=0
MOVL C00939 V=800.0 PL=0
MOVL C00940 V=800.0 PL=0
MOVL C00941 V=800.0 PL=0
MOVL C00942 V=800.0 PL=0
MOVL C00943 V=800.0 PL=0
MOVL C00944 V=800.0 PL=0
MOVL C00945 V=800.0 PL=0
MOVL C00946 V=800.0 PL=0
MOVL C00947 V=800.0 PL=0
MOVL C00948 V=800.0 PL=0
MOVL C00949 V=800.0 PL=0
MOVL C00950 V=800.0 PL=0
MOVL C00951 V=800.0 PL=0
MOVL C00952 V=800.0 PL=0
MOVL C00953 V=800.0 PL=0
MOVL C00954 V=800.0 PL=0
MOVL C00955 V=800.0 PL=0
MOVL C00956 V=800.0 PL=0
MOVL C00957 V=800.0 PL=0
MOVL C00958 V=800.0 PL=0
MOVL C00959 V=800.0 PL=0
MOVL C00960 V=800.0 PL=0
MOVL C00961 V=800.0 PL=0
MOVL C00962 V=800.0 PL=0
MOVL C00963 V=800.0 PL=0
MOVL C00964 V=800.0 PL=0
MOVL C00965 V=800.0 PL=0
MOVL C00966 V=800.0 PL=0
MOVL C00967 V=800.0 PL=0
MOVL C00968 V=800.0 PL=0
MOVL C00969 V=800.0 PL=0
MOVL C00970 V=800.0 PL=0
MOVL C00971 V=800.0 PL=0
MOVL C00972 V=800.0 PL=0
MOVL C00973 V=800.0 PL=0
MOVL C00974 V=800.0 PL=0
MOVL C00975 V=800.0 PL=0
MOVL C00976 V=800.0 PL=0
MOVL C00977 V=800.0 PL=0
MOVL C00978 V=800.0 PL=0
MOVL C00979 V=800.0 PL=0
MOVL C00980 V=800.0 PL=0
MOVL C00981 V=800.0 PL=0
MOVL C00982 V=800.0 PL=0
MOVL C00983 V=800.0 PL=0
MOVL C00984 V=800.0 PL=0
MOVL C00985 V=800.0 PL=0
MOVL C00986 V=800.0 PL=0
MOVL C00987 V=800.0 PL=0
MOVL C00988 V=800.0 PL=0
MOVL C00989 V=800.0 PL=0
MOVL C00990 V=800.0 PL=0
MOVL C00991 V=800.0 PL=0
MOVL C00992 V=800.0 PL=0
MOVL C00993 V=800.0 PL=0
MOVL C00994 V=800.0 PL=0
MOVL C00995 V=800.0 PL=0
MOVL C00996 V=800.0 PL=0
MOVL C00997 V=800.0 PL=0
MOVL C00998 V=800.0 PL=0
MOVL C00999 V=800.0 PL=0
MOVL C01000 V=800.0 PL=0
MOVL C01001 V=800.0 PL=0
MOVL C01002 V=800.0 PL=0
MOVL C01003 V=800.0 PL=0
MOVL C01004 V=800.0 PL=0
MOVL C01005 V=800.0 PL=0
MOVL C01006 V=800.0 PL=0
MOVL C01007 V=800.0 PL=0
MOVL C01008 V=800.0 PL=0
MOVL C01009 V=800.0 PL=0
MOVL C01010 V=800.0 PL=0
MOVL C01011 V=800.0 PL=0
MOVL C01012 V=800.0 PL=0
MOVL C01013 V=800.0 PL=0
MOVL C01014 V=800.0 PL=0
MOVL C01015 V=800.0 PL=0
MOVL C01016 V=800.0 PL=0
MOVL C01017 V=800.0 PL=0
MOVL C01018 V=800.0 PL=0
MOVL C01019 V=800.0 PL=0
MOVL C01020 V=800.0 PL=0
MOVL C01021 V=800.0 PL=0
MOVL C01022 V=800.0 PL=0
MOVL C01023 V=800.0 PL=0
MOVL C01024 V=800.0 PL=0
MOVL C01025 V=800.0 PL=0
MOVL C01026 V=800.0 PL=0
MOVL C01027 V=800.0 PL=0
MOVL C01028 V=800.0 PL=0
MOVL C01029 V=800.0 PL=0
MOVL C01030 V=800.0 PL=0
MOVL C01031 V=800.0 PL=0
MOVL C01032 V=800.0 PL=0
MOVL C01033 V=800.0 PL=0
MOVL C01034 V=800.0 PL=0
MOVL C01035 V=800.0 PL=0
MOVL C01036 V=800.0 PL=0
MOVL C01037 V=800.0 PL=0
MOVL C01038 V=800.0 PL=0
MOVL C01039 V=800.0 PL=0
MOVL C01040 V=800.0 PL=0
MOVL C01041 V=800.0 PL=0
MOVL C01042 V=800.0 PL=0
MOVL C01043 V=800.0 PL=0
MOVL C01044 V=800.0 PL=0
MOVL C01045 V=800.0 PL=0
MOVL C01046 V=800.0 PL=0
MOVL C01047 V=800.0 PL=0
MOVL C01048 V=800.0 PL=0
MOVL C01049 V=800.0 PL=0
MOVL C01050 V=800.0 PL=0
MOVL C01051 V=800.0 PL=0
MOVL C01052 V=800.0 PL=0
MOVL C01053 V=800.0 PL=0
MOVL C01054 V=800.0 PL=0
MOVL C01055 V=800.0 PL=0
MOVL C01056 V=800.0 PL=0
MOVL C01057 V=800.0 PL=0
MOVL C01058 V=800.0 PL=0
MOVL C01059 V=800.0 PL=0
MOVL C01060 V=800.0 PL=0
MOVL C01061 V=800.0 PL=0
MOVL C01062 V=800.0 PL=0
MOVL C01063 V=800.0 PL=0
MOVL C01064 V=800.0 PL=0
MOVL C01065 V=800.0 PL=0
MOVL C01066 V=800.0 PL=0
MOVL C01067 V=800.0 PL=0
MOVL C01068 V=800.0 PL=0
MOVL C01069 V=800.0 PL=0
MOVL C01070 V=800.0 PL=0
MOVL C01071 V=800.0 PL=0
MOVL C01072 V=800.0 PL=0
MOVL C01073 V=800.0 PL=0
MOVL C01074 V=800.0 PL=0
MOVL C01075 V=800.0 PL=0
MOVL C01076 V=800.0 PL=0
MOVL C01077 V=800.0 PL=0
MOVL C01078 V=800.0 PL=0
MOVL C01079 V=800.0 PL=0
MOVL C01080 V=800.0 PL=0
MOVL C01081 V=800.0 PL=0
MOVL C01082 V=800.0 PL=0
MOVL C01083 V=800.0 PL=0
MOVL C01084 V=800.0 PL=0
MOVL C01085 V=800.0 PL=0
MOVL C01086 V=800.0 PL=0
MOVL C01087 V=800.0 PL=0
MOVL C01088 V=800.0 PL=0
MOVL C01089 V=800.0 PL=0
MOVL C01090 V=800.0 PL=0
MOVL C01091 V=800.0 PL=0
MOVL C01092 V=800.0 PL=0
MOVL C01093 V=800.0 PL=0
MOVL C01094 V=800.0 PL=0
MOVL C01095 V=800.0 PL=0
MOVL C01096 V=800.0 PL=0
MOVL C01097 V=800.0 PL=0
MOVL C01098 V=800.0 PL=0
MOVL C01099 V=800.0 PL=0
MOVL C01100 V=800.0 PL=0
MOVL C01101 V=800.0 PL=0
MOVL C01102 V=800.0 PL=0
MOVL C01103 V=800.0 PL=0
MOVL C01104 V=800.0 PL=0
MOVL C01105 V=800.0 PL=0
MOVL C01106 V=800.0 PL=0
MOVL C01107 V=800.0 PL=0
MOVL C01108 V=800.0 PL=0
MOVL C01109 V=800.0 PL=0
MOVL C01110 V=800.0 PL=0
MOVL C01111 V=800.0 PL=0
MOVL C01112 V=800.0 PL=0
MOVL C01113 V=800.0 PL=0
MOVL C01114 V=800.0 PL=0
MOVL C01115 V=800.0 PL=0
MOVL C01116 V=800.0 PL=0
MOVL C01117 V=800.0 PL=0
MOVL C01118 V=800.0 PL=0
MOVL C01119 V=800.0 PL=0
MOVL C01120 V=800.0 PL=0
MOVL C01121 V=800.0 PL=0
MOVL C01122 V=800.0 PL=0
MOVL C01123 V=800.0 PL=0
MOVL C01124 V=800.0 PL=0
MOVL C01125 V=800.0 PL=0
MOVL C01126 V=800.0 PL=0
MOVL C01127 V=800.0 PL=0
MOVL C01128 V=800.0 PL=0
MOVL C01129 V=800.0 PL=0
MOVL C01130 V=800.0 PL=0
MOVL C01131 V=800.0 PL=0
MOVL C01132 V=800.0 PL=0
MOVL C01133 V=800.0 PL=0
MOVL C01134 V=800.0 PL=0
MOVL C01135 V=800.0 PL=0
MOVL C01136 V=800.0 PL=0
MOVL C01137 V=800.0 PL=0
MOVL C01138 V=800.0 PL=0
MOVL C01139 V=800.0 PL=0
MOVL C01140 V=800.0 PL=0
MOVL C01141 V=800.0 PL=0
MOVL C01142 V=800.0 PL=0
MOVL C01143 V=800.0 PL=0
MOVL C01144 V=800.0 PL=0
MOVL C01145 V=800.0 PL=0
MOVL C01146 V=800.0 PL=0
MOVL C01147 V=800.0 PL=0
MOVL C01148 V=800.0 PL=0
MOVL C01149 V=800.0 PL=0
MOVL C01150 V=800.0 PL=0
MOVL C01151 V=800.0 PL=0
MOVL C01152 V=800.0 PL=0
MOVL C01153 V=800.0 PL=0
MOVL C01154 V=800.0 PL=0
MOVL C01155 V=800.0 PL=0
MOVL C01156 V=800.0 PL=0
MOVL C01157 V=800.0 PL=0
MOVL C01158 V=800.0 PL=0
MOVL C01159 V=800.0 PL=0
MOVL C01160 V=800.0 PL=0
MOVL C01161 V=800.0 PL=0
MOVL C01162 V=800.0 PL=0
MOVL C01163 V=800.0 PL=0
MOVL C01164 V=800.0 PL=0
MOVL C01165 V=800.0 PL=0
MOVL C01166 V=800.0 PL=0
MOVL C01167 V=800.0 PL=0
MOVL C01168 V=800.0 PL=0
MOVL C01169 V=800.0 PL=0
MOVL C01170 V=800.0 PL=0
MOVL C01171 V=800.0 PL=0
MOVL C01172 V=800.0 PL=0
MOVL C01173 V=800.0 PL=0
MOVL C01174 V=800.0 PL=0
MOVL C01175 V=800.0 PL=0
MOVL C01176 V=800.0 PL=0
MOVL C01177 V=800.0 PL=0
MOVL C01178 V=800.0 PL=0
MOVL C01179 V=800.0 PL=0
MOVL C01180 V=800.0 PL=0
MOVL C01181 V=800.0 PL=0
MOVL C01182 V=800.0 PL=0
MOVL C01183 V=800.0 PL=0
MOVL C01184 V=800.0 PL=0
MOVL C01185 V=800.0 PL=0
MOVL C01186 V=800.0 PL=0
MOVL C01187 V=800.0 PL=0
MOVL C01188 V=800.0 PL=0
MOVL C01189 V=800.0 PL=0
MOVL C01190 V=800.0 PL=0
MOVL C01191 V=800.0 PL=0
MOVL C01192 V=800.0 PL=0
MOVL C01193 V=800.0 PL=0
MOVL C01194 V=800.0 PL=0
MOVL C01195 V=800.0 PL=0
MOVL C01196 V=800.0 PL=0
MOVL C01197 V=800.0 PL=0
MOVL C01198 V=800.0 PL=0
MOVL C01199 V=800.0 PL=0
MOVL C01200 V=800.0 PL=0
MOVL C01201 V=800.0 PL=0
MOVL C01202 V=800.0 PL=0
MOVL C01203 V=800.0 PL=0
MOVL C01204 V=800.0 PL=0
MOVL C01205 V=800.0 PL=0
MOVL C01206 V=800.0 PL=0
MOVL C01207 V=800.0 PL=0
MOVL C01208 V=800.0 PL=0
MOVL C01209 V=800.0 PL=0
MOVL C01210 V=800.0 PL=0
MOVL C01211 V=800.0 PL=0
MOVL C01212 V=800.0 PL=0
MOVL C01213 V=800.0 PL=0
MOVL C01214 V=800.0 PL=0
MOVL C01215 V=800.0 PL=0
MOVL C01216 V=800.0 PL=0
MOVL C01217 V=800.0 PL=0
MOVL C01218 V=800.0 PL=0
MOVL C01219 V=800.0 PL=0
MOVL C01220 V=800.0 PL=0
MOVL C01221 V=800.0 PL=0
MOVL C01222 V=800.0 PL=0
MOVL C01223 V=800.0 PL=0
MOVL C01224 V=800.0 PL=0
MOVL C01225 V=800.0 PL=0
MOVL C01226 V=800.0 PL=0
MOVL C01227 V=800.0 PL=0
MOVL C01228 V=800.0 PL=0
MOVL C01229 V=800.0 PL=0
MOVL C01230 V=800.0 PL=0
MOVL C01231 V=800.0 PL=0
MOVL C01232 V=800.0 PL=0
MOVL C01233 V=800.0 PL=0
MOVL C01234 V=800.0 PL=0
MOVL C01235 V=800.0 PL=0
MOVL C01236 V=800.0 PL=0
MOVL C01237 V=800.0 PL=0
MOVL C01238 V=800.0 PL=0
MOVL C01239 V=800.0 PL=0
MOVL C01240 V=800.0 PL=0
MOVL C01241 V=800.0 PL=0
MOVL C01242 V=800.0 PL=0
MOVL C01243 V=800.0 PL=0
MOVL C01244 V=800.0 PL=0
MOVL C01245 V=800.0 PL=0
MOVL C01246 V=800.0 PL=0
MOVL C01247 V=800.0 PL=0
MOVL C01248 V=800.0 PL=0
MOVL C01249 V=800.0 PL=0
MOVL C01250 V=800.0 PL=0
MOVL C01251 V=800.0 PL=0
MOVL C01252 V=800.0 PL=0
MOVL C01253 V=800.0 PL=0
MOVL C01254 V=800.0 PL=0
MOVL C01255 V=800.0 PL=0
MOVL C01256 V=800.0 PL=0
MOVL C01257 V=800.0 PL=0
MOVL C01258 V=800.0 PL=0
MOVL C01259 V=800.0 PL=0
MOVL C01260 V=800.0 PL=0
MOVL C01261 V=800.0 PL=0
MOVL C01262 V=800.0 PL=0
MOVL C01263 V=800.0 PL=0
MOVL C01264 V=800.0 PL=0
MOVL C01265 V=800.0 PL=0
MOVL C01266 V=800.0 PL=0
MOVL C01267 V=800.0 PL=0
MOVL C01268 V=800.0 PL=0
MOVL C01269 V=800.0 PL=0
MOVL C01270 V=800.0 PL=0
MOVL C01271 V=800.0 PL=0
MOVL C01272 V=800.0 PL=0
MOVL C01273 V=800.0 PL=0
MOVL C01274 V=800.0 PL=0
MOVL C01275 V=800.0 PL=0
MOVL C01276 V=800.0 PL=0
MOVL C01277 V=800.0 PL=0
MOVL C01278 V=800.0 PL=0
MOVL C01279 V=800.0 PL=0
MOVL C01280 V=800.0 PL=0
MOVL C01281 V=800.0 PL=0
MOVL C01282 V=800.0 PL=0
MOVL C01283 V=800.0 PL=0
MOVL C01284 V=800.0 PL=0
MOVL C01285 V=800.0 PL=0
MOVL C01286 V=800.0 PL=0
MOVL C01287 V=800.0 PL=0
MOVL C01288 V=800.0 PL=0
MOVL C01289 V=800.0 PL=0
MOVL C01290 V=800.0 PL=0
MOVL C01291 V=800.0 PL=0
MOVL C01292 V=800.0 PL=0
MOVL C01293 V=800.0 PL=0
MOVL C01294 V=800.0 PL=0
MOVL C01295 V=800.0 PL=0
MOVL C01296 V=800.0 PL=0
MOVL C01297 V=800.0 PL=0
MOVL C01298 V=800.0 PL=0
MOVL C01299 V=800.0 PL=0
MOVL C01300 V=800.0 PL=0
MOVL C01301 V=800.0 PL=0
MOVL C01302 V=800.0 PL=0
MOVL C01303 V=800.0 PL=0
MOVL C01304 V=800.0 PL=0
MOVL C01305 V=800.0 PL=0
MOVL C01306 V=800.0 PL=0
MOVL C01307 V=800.0 PL=0
MOVL C01308 V=800.0 PL=0
MOVL C01309 V=800.0 PL=0
MOVL C01310 V=800.0 PL=0
MOVL C01311 V=800.0 PL=0
MOVL C01312 V=800.0 PL=0
MOVL C01313 V=800.0 PL=0
MOVL C01314 V=800.0 PL=0
MOVL C01315 V=800.0 PL=0
MOVL C01316 V=800.0 PL=0
MOVL C01317 V=800.0 PL=0
MOVL C01318 V=800.0 PL=0
MOVL C01319 V=800.0 PL=0
MOVL C01320 V=800.0 PL=0
MOVL C01321 V=800.0 PL=0
MOVL C01322 V=800.0 PL=0
MOVL C01323 V=800.0 PL=0
MOVL C01324 V=800.0 PL=0
MOVL C01325 V=800.0 PL=0
MOVL C01326 V=800.0 PL=0
MOVL C01327 V=800.0 PL=0
MOVL C01328 V=800.0 PL=0
MOVL C01329 V=800.0 PL=0
MOVL C01330 V=800.0 PL=0
MOVL C01331 V=800.0 PL=0
MOVL C01332 V=800.0 PL=0
MOVL C01333 V=800.0 PL=0
MOVL C01334 V=800.0 PL=0
MOVL C01335 V=800.0 PL=0
MOVL C01336 V=800.0 PL=0
MOVL C01337 V=800.0 PL=0
MOVL C01338 V=800.0 PL=0
MOVL C01339 V=800.0 PL=0
MOVL C01340 V=800.0 PL=0
MOVL C01341 V=800.0 PL=0
MOVL C01342 V=800.0 PL=0
MOVL C01343 V=800.0 PL=0
MOVL C01344 V=800.0 PL=0
MOVL C01345 V=800.0 PL=0
MOVL C01346 V=800.0 PL=0
MOVL C01347 V=800.0 PL=0
MOVL C01348 V=800.0 PL=0
MOVL C01349 V=800.0 PL=0
MOVL C01350 V=800.0 PL=0
MOVL C01351 V=800.0 PL=0
MOVL C01352 V=800.0 PL=0
MOVL C01353 V=800.0 PL=0
MOVL C01354 V=800.0 PL=0
MOVL C01355 V=800.0 PL=0
MOVL C01356 V=800.0 PL=0
MOVL C01357 V=800.0 PL=0
MOVL C01358 V=800.0 PL=0
MOVL C01359 V=800.0 PL=0
MOVL C01360 V=800.0 PL=0
MOVL C01361 V=800.0 PL=0
MOVL C01362 V=800.0 PL=0
MOVL C01363 V=800.0 PL=0
MOVL C01364 V=800.0 PL=0
MOVL C01365 V=800.0 PL=0
MOVL C01366 V=800.0 PL=0
MOVL C01367 V=800.0 PL=0
MOVL C01368 V=800.0 PL=0
MOVL C01369 V=800.0 PL=0
MOVL C01370 V=800.0 PL=0
MOVL C01371 V=800.0 PL=0
MOVL C01372 V=800.0 PL=0
MOVL C01373 V=800.0 PL=0
MOVL C01374 V=800.0 PL=0
MOVL C01375 V=800.0 PL=0
MOVL C01376 V=800.0 PL=0
MOVL C01377 V=800.0 PL=0
MOVL C01378 V=800.0 PL=0
MOVL C01379 V=800.0 PL=0
MOVL C01380 V=800.0 PL=0
MOVL C01381 V=800.0 PL=0
MOVL C01382 V=800.0 PL=0
MOVL C01383 V=800.0 PL=0
MOVL C01384 V=800.0 PL=0
MOVL C01385 V=800.0 PL=0
MOVL C01386 V=800.0 PL=0
MOVL C01387 V=800.0 PL=0
MOVL C01388 V=800.0 PL=0
MOVL C01389 V=800.0 PL=0
MOVL C01390 V=800.0 PL=0
MOVL C01391 V=800.0 PL=0
MOVL C01392 V=800.0 PL=0
MOVL C01393 V=800.0 PL=0
MOVL C01394 V=800.0 PL=0
MOVL C01395 V=800.0 PL=0
MOVL C01396 V=800.0 PL=0
MOVL C01397 V=800.0 PL=0
MOVL C01398 V=800.0 PL=0
MOVL C01399 V=800.0 PL=0
MOVL C01400 V=800.0 PL=0
MOVL C01401 V=800.0 PL=0
MOVL C01402 V=800.0 PL=0
MOVL C01403 V=800.0 PL=0
MOVL C01404 V=800.0 PL=0
MOVL C01405 V=800.0 PL=0
MOVL C01406 V=800.0 PL=0
MOVL C01407 V=800.0 PL=0
MOVL C01408 V=800.0 PL=0
MOVL C01409 V=800.0 PL=0
MOVL C01410 V=800.0 PL=0
MOVL C01411 V=800.0 PL=0
MOVL C01412 V=800.0 PL=0
MOVL C01413 V=800.0 PL=0
MOVL C01414 V=800.0 PL=0
MOVL C01415 V=800.0 PL=0
MOVL C01416 V=800.0 PL=0
MOVL C01417 V=800.0 PL=0
MOVL C01418 V=800.0 PL=0
MOVL C01419 V=800.0 PL=0
MOVL C01420 V=800.0 PL=0
MOVL C01421 V=800.0 PL=0
MOVL C01422 V=800.0 PL=0
MOVL C01423 V=800.0 PL=0
MOVL C01424 V=800.0 PL=0
MOVL C01425 V=800.0 PL=0
MOVL C01426 V=800.0 PL=0
MOVL C01427 V=800.0 PL=0
MOVL C01428 V=800.0 PL=0
MOVL C01429 V=800.0 PL=0
MOVL C01430 V=800.0 PL=0
MOVL C01431 V=800.0 PL=0
MOVL C01432 V=800.0 PL=0
MOVL C01433 V=800.0 PL=0
MOVL C01434 V=800.0 PL=0
MOVL C01435 V=800.0 PL=0
MOVL C01436 V=800.0 PL=0
MOVL C01437 V=800.0 PL=0
MOVL C01438 V=800.0 PL=0
MOVL C01439 V=800.0 PL=0
MOVL C01440 V=800.0 PL=0
MOVL C01441 V=800.0 PL=0
MOVL C01442 V=800.0 PL=0
MOVL C01443 V=800.0 PL=0
MOVL C01444 V=800.0 PL=0
MOVL C01445 V=800.0 PL=0
MOVL C01446 V=800.0 PL=0
MOVL C01447 V=800.0 PL=0
MOVL C01448 V=800.0 PL=0
MOVL C01449 V=800.0 PL=0
MOVL C01450 V=800.0 PL=0
MOVL C01451 V=800.0 PL=0
MOVL C01452 V=800.0 PL=0
MOVL C01453 V=800.0 PL=0
MOVL C01454 V=800.0 PL=0
MOVL C01455 V=800.0 PL=0
MOVL C01456 V=800.0 PL=0
MOVL C01457 V=800.0 PL=0
MOVL C01458 V=800.0 PL=0
MOVL C01459 V=800.0 PL=0
MOVL C01460 V=800.0 PL=0
MOVL C01461 V=800.0 PL=0
MOVL C01462 V=800.0 PL=0
MOVL C01463 V=800.0 PL=0
MOVL C01464 V=800.0 PL=0
MOVL C01465 V=800.0 PL=0
MOVL C01466 V=800.0 PL=0
MOVL C01467 V=800.0 PL=0
MOVL C01468 V=800.0 PL=0
MOVL C01469 V=800.0 PL=0
MOVL C01470 V=800.0 PL=0
MOVL C01471 V=800.0 PL=0
MOVL C01472 V=800.0 PL=0
MOVL C01473 V=800.0 PL=0
MOVL C01474 V=800.0 PL=0
MOVL C01475 V=800.0 PL=0
MOVL C01476 V=800.0 PL=0
MOVL C01477 V=800.0 PL=0
MOVL C01478 V=800.0 PL=0
MOVL C01479 V=800.0 PL=0
MOVL C01480 V=800.0 PL=0
MOVL C01481 V=800.0 PL=0
MOVL C01482 V=800.0 PL=0
MOVL C01483 V=800.0 PL=0
MOVL C01484 V=800.0 PL=0
MOVL C01485 V=800.0 PL=0
MOVL C01486 V=800.0 PL=0
MOVL C01487 V=800.0 PL=0
MOVL C01488 V=800.0 PL=0
MOVL C01489 V=800.0 PL=0
MOVL C01490 V=800.0 PL=0
MOVL C01491 V=800.0 PL=0
MOVL C01492 V=800.0 PL=0
MOVL C01493 V=800.0 PL=0
MOVL C01494 V=800.0 PL=0
MOVL C01495 V=800.0 PL=0
MOVL C01496 V=800.0 PL=0
MOVL C01497 V=800.0 PL=0
MOVL C01498 V=800.0 PL=0
MOVL C01499 V=800.0 PL=0
MOVL C01500 V=800.0 PL=0
MOVL C01501 V=800.0 PL=0
MOVL C01502 V=800.0 PL=0
MOVL C01503 V=800.0 PL=0
MOVL C01504 V=800.0 PL=0
MOVL C01505 V=800.0 PL=0
MOVL C01506 V=800.0 PL=0
MOVL C01507 V=800.0 PL=0
MOVL C01508 V=800.0 PL=0
MOVL C01509 V=800.0 PL=0
MOVL C01510 V=800.0 PL=0
MOVL C01511 V=800.0 PL=0
MOVL C01512 V=800.0 PL=0
MOVL C01513 V=800.0 PL=0
MOVL C01514 V=800.0 PL=0
MOVL C01515 V=800.0 PL=0
MOVL C01516 V=800.0 PL=0
MOVL C01517 V=800.0 PL=0
MOVL C01518 V=800.0 PL=0
MOVL C01519 V=800.0 PL=0
MOVL C01520 V=800.0 PL=0
MOVL C01521 V=800.0 PL=0
MOVL C01522 V=800.0 PL=0
MOVL C01523 V=800.0 PL=0
MOVL C01524 V=800.0 PL=0
MOVL C01525 V=800.0 PL=0
MOVL C01526 V=800.0 PL=0
MOVL C01527 V=800.0 PL=0
MOVL C01528 V=800.0 PL=0
MOVL C01529 V=800.0 PL=0
MOVL C01530 V=800.0 PL=0
MOVL C01531 V=800.0 PL=0
MOVL C01532 V=800.0 PL=0
MOVL C01533 V=800.0 PL=0
MOVL C01534 V=800.0 PL=0
MOVL C01535 V=800.0 PL=0
MOVL C01536 V=800.0 PL=0
MOVL C01537 V=800.0 PL=0
MOVL C01538 V=800.0 PL=0
MOVL C01539 V=800.0 PL=0
MOVL C01540 V=800.0 PL=0
MOVL C01541 V=800.0 PL=0
MOVL C01542 V=800.0 PL=0
MOVL C01543 V=800.0 PL=0
MOVL C01544 V=800.0 PL=0
MOVL C01545 V=800.0 PL=0
MOVL C01546 V=800.0 PL=0
MOVL C01547 V=800.0 PL=0
MOVL C01548 V=800.0 PL=0
MOVL C01549 V=800.0 PL=0
MOVL C01550 V=800.0 PL=0
MOVL C01551 V=800.0 PL=0
MOVL C01552 V=800.0 PL=0
MOVL C01553 V=800.0 PL=0
MOVL C01554 V=800.0 PL=0
MOVL C01555 V=800.0 PL=0
MOVL C01556 V=800.0 PL=0
MOVL C01557 V=800.0 PL=0
MOVL C01558 V=800.0 PL=0
MOVL C01559 V=800.0 PL=0
MOVL C01560 V=800.0 PL=0
MOVL C01561 V=800.0 PL=0
MOVL C01562 V=800.0 PL=0
MOVL C01563 V=800.0 PL=0
MOVL C01564 V=800.0 PL=0
MOVL C01565 V=800.0 PL=0
MOVL C01566 V=800.0 PL=0
MOVL C01567 V=800.0 PL=0
MOVL C01568 V=800.0 PL=0
MOVL C01569 V=800.0 PL=0
MOVL C01570 V=800.0 PL=0
MOVL C01571 V=800.0 PL=0
MOVL C01572 V=800.0 PL=0
MOVL C01573 V=800.0 PL=0
MOVL C01574 V=800.0 PL=0
MOVL C01575 V=800.0 PL=0
MOVL C01576 V=800.0 PL=0
MOVL C01577 V=800.0 PL=0
MOVL C01578 V=800.0 PL=0
MOVL C01579 V=800.0 PL=0
MOVL C01580 V=800.0 PL=0
MOVL C01581 V=800.0 PL=0
MOVL C01582 V=800.0 PL=0
MOVL C01583 V=800.0 PL=0
MOVL C01584 V=800.0 PL=0
MOVL C01585 V=800.0 PL=0
MOVL C01586 V=800.0 PL=0
MOVL C01587 V=800.0 PL=0
MOVL C01588 V=800.0 PL=0
MOVL C01589 V=800.0 PL=0
MOVL C01590 V=800.0 PL=0
MOVL C01591 V=800.0 PL=0
MOVL C01592 V=800.0 PL=0
MOVL C01593 V=800.0 PL=0
MOVL C01594 V=800.0 PL=0
MOVL C01595 V=800.0 PL=0
MOVL C01596 V=800.0 PL=0
MOVL C01597 V=800.0 PL=0
MOVL C01598 V=800.0 PL=0
MOVL C01599 V=800.0 PL=0
MOVL C01600 V=800.0 PL=0
MOVL C01601 V=800.0 PL=0
MOVL C01602 V=800.0 PL=0
MOVL C01603 V=800.0 PL=0
MOVL C01604 V=800.0 PL=0
MOVL C01605 V=800.0 PL=0
MOVL C01606 V=800.0 PL=0
MOVL C01607 V=800.0 PL=0
MOVL C01608 V=800.0 PL=0
MOVL C01609 V=800.0 PL=0
MOVL C01610 V=800.0 PL=0
MOVL C01611 V=800.0 PL=0
MOVL C01612 V=800.0 PL=0
MOVL C01613 V=800.0 PL=0
MOVL C01614 V=800.0 PL=0
MOVL C01615 V=800.0 PL=0
MOVL C01616 V=800.0 PL=0
MOVL C01617 V=800.0 PL=0
MOVL C01618 V=800.0 PL=0
MOVL C01619 V=800.0 PL=0
MOVL C01620 V=800.0 PL=0
MOVL C01621 V=800.0 PL=0
MOVL C01622 V=800.0 PL=0
MOVL C01623 V=800.0 PL=0
MOVL C01624 V=800.0 PL=0
MOVL C01625 V=800.0 PL=0
MOVL C01626 V=800.0 PL=0
MOVL C01627 V=800.0 PL=0
MOVL C01628 V=800.0 PL=0
MOVL C01629 V=800.0 PL=0
MOVL C01630 V=800.0 PL=0
MOVL C01631 V=800.0 PL=0
MOVL C01632 V=800.0 PL=0
MOVL C01633 V=800.0 PL=0
MOVL C01634 V=800.0 PL=0
MOVL C01635 V=800.0 PL=0
MOVL C01636 V=800.0 PL=0
MOVL C01637 V=800.0 PL=0
MOVL C01638 V=800.0 PL=0
MOVL C01639 V=800.0 PL=0
MOVL C01640 V=800.0 PL=0
MOVL C01641 V=800.0 PL=0
MOVL C01642 V=800.0 PL=0
MOVL C01643 V=800.0 PL=0
MOVL C01644 V=800.0 PL=0
MOVL C01645 V=800.0 PL=0
MOVL C01646 V=800.0 PL=0
MOVL C01647 V=800.0 PL=0
MOVL C01648 V=800.0 PL=0
MOVL C01649 V=800.0 PL=0
MOVL C01650 V=800.0 PL=0
MOVL C01651 V=800.0 PL=0
MOVL C01652 V=800.0 PL=0
MOVL C01653 V=800.0 PL=0
MOVL C01654 V=800.0 PL=0
MOVL C01655 V=800.0 PL=0
MOVL C01656 V=800.0 PL=0
MOVL C01657 V=800.0 PL=0
MOVL C01658 V=800.0 PL=0
MOVL C01659 V=800.0 PL=0
MOVL C01660 V=800.0 PL=0
MOVL C01661 V=800.0 PL=0
MOVL C01662 V=800.0 PL=0
MOVL C01663 V=800.0 PL=0
MOVL C01664 V=800.0 PL=0
MOVL C01665 V=800.0 PL=0
MOVL C01666 V=800.0 PL=0
MOVL C01667 V=800.0 PL=0
MOVL C01668 V=800.0 PL=0
MOVL C01669 V=800.0 PL=0
MOVL C01670 V=800.0 PL=0
MOVL C01671 V=800.0 PL=0
MOVL C01672 V=800.0 PL=0
MOVL C01673 V=800.0 PL=0
MOVL C01674 V=800.0 PL=0
MOVL C01675 V=800.0 PL=0
MOVL C01676 V=800.0 PL=0
MOVL C01677 V=800.0 PL=0
MOVL C01678 V=800.0 PL=0
MOVL C01679 V=800.0 PL=0
MOVL C01680 V=800.0 PL=0
MOVL C01681 V=800.0 PL=0
MOVL C01682 V=800.0 PL=0
MOVL C01683 V=800.0 PL=0
MOVL C01684 V=800.0 PL=0
MOVL C01685 V=800.0 PL=0
MOVL C01686 V=800.0 PL=0
MOVL C01687 V=800.0 PL=0
MOVL C01688 V=800.0 PL=0
MOVL C01689 V=800.0 PL=0
MOVL C01690 V=800.0 PL=0
MOVL C01691 V=800.0 PL=0
MOVL C01692 V=800.0 PL=0
MOVL C01693 V=800.0 PL=0
MOVL C01694 V=800.0 PL=0
MOVL C01695 V=800.0 PL=0
MOVL C01696 V=800.0 PL=0
MOVL C01697 V=800.0 PL=0
MOVL C01698 V=800.0 PL=0
MOVL C01699 V=800.0 PL=0
MOVL C01700 V=800.0 PL=0
MOVL C01701 V=800.0 PL=0
MOVL C01702 V=800.0 PL=0
MOVL C01703 V=800.0 PL=0
MOVL C01704 V=800.0 PL=0
MOVL C01705 V=800.0 PL=0
MOVL C01706 V=800.0 PL=0
MOVL C01707 V=800.0 PL=0
MOVL C01708 V=800.0 PL=0
MOVL C01709 V=800.0 PL=0
MOVL C01710 V=800.0 PL=0
MOVL C01711 V=800.0 PL=0
MOVL C01712 V=800.0 PL=0
MOVL C01713 V=800.0 PL=0
MOVL C01714 V=800.0 PL=0
MOVL C01715 V=800.0 PL=0
MOVL C01716 V=800.0 PL=0
MOVL C01717 V=800.0 PL=0
MOVL C01718 V=800.0 PL=0
MOVL C01719 V=800.0 PL=0
MOVL C01720 V=800.0 PL=0
MOVL C01721 V=800.0 PL=0
MOVL C01722 V=800.0 PL=0
MOVL C01723 V=800.0 PL=0
MOVL C01724 V=800.0 PL=0
MOVL C01725 V=800.0 PL=0
MOVL C01726 V=800.0 PL=0
MOVL C01727 V=800.0 PL=0
MOVL C01728 V=800.0 PL=0
MOVL C01729 V=800.0 PL=0
MOVL C01730 V=800.0 PL=0
MOVL C01731 V=800.0 PL=0
MOVL C01732 V=800.0 PL=0
MOVL C01733 V=800.0 PL=0
MOVL C01734 V=800.0 PL=0
MOVL C01735 V=800.0 PL=0
MOVL C01736 V=800.0 PL=0
MOVL C01737 V=800.0 PL=0
MOVL C01738 V=800.0 PL=0
MOVL C01739 V=800.0 PL=0
MOVL C01740 V=800.0 PL=0
MOVL C01741 V=800.0 PL=0
MOVL C01742 V=800.0 PL=0
MOVL C01743 V=800.0 PL=0
MOVL C01744 V=800.0 PL=0
MOVL C01745 V=800.0 PL=0
MOVL C01746 V=800.0 PL=0
MOVL C01747 V=800.0 PL=0
MOVL C01748 V=800.0 PL=0
MOVL C01749 V=800.0 PL=0
MOVL C01750 V=800.0 PL=0
MOVL C01751 V=800.0 PL=0
MOVL C01752 V=800.0 PL=0
MOVL C01753 V=800.0 PL=0
MOVL C01754 V=800.0 PL=0
MOVL C01755 V=800.0 PL=0
MOVL C01756 V=800.0 PL=0
MOVL C01757 V=800.0 PL=0
MOVL C01758 V=800.0 PL=0
MOVL C01759 V=800.0 PL=0
MOVL C01760 V=800.0 PL=0
MOVL C01761 V=800.0 PL=0
MOVL C01762 V=800.0 PL=0
MOVL C01763 V=800.0 PL=0
MOVL C01764 V=800.0 PL=0
MOVL C01765 V=800.0 PL=0
MOVL C01766 V=800.0 PL=0
MOVL C01767 V=800.0 PL=0
MOVL C01768 V=800.0 PL=0
MOVL C01769 V=800.0 PL=0
MOVL C01770 V=800.0 PL=0
MOVL C01771 V=800.0 PL=0
MOVL C01772 V=800.0 PL=0
MOVL C01773 V=800.0 PL=0
MOVL C01774 V=800.0 PL=0
MOVL C01775 V=800.0 PL=0
MOVL C01776 V=800.0 PL=0
MOVL C01777 V=800.0 PL=0
MOVL C01778 V=800.0 PL=0
MOVL C01779 V=800.0 PL=0
MOVL C01780 V=800.0 PL=0
MOVL C01781 V=800.0 PL=0
MOVL C01782 V=800.0 PL=0
MOVL C01783 V=800.0 PL=0
MOVL C01784 V=800.0 PL=0
MOVL C01785 V=800.0 PL=0
MOVL C01786 V=800.0 PL=0
MOVL C01787 V=800.0 PL=0
MOVL C01788 V=800.0 PL=0
MOVL C01789 V=800.0 PL=0
MOVL C01790 V=800.0 PL=0
MOVL C01791 V=800.0 PL=0
MOVL C01792 V=800.0 PL=0
MOVL C01793 V=800.0 PL=0
MOVL C01794 V=800.0 PL=0
MOVL C01795 V=800.0 PL=0
MOVL C01796 V=800.0 PL=0
MOVL C01797 V=800.0 PL=0
MOVL C01798 V=800.0 PL=0
MOVL C01799 V=800.0 PL=0
MOVL C01800 V=800.0 PL=0
MOVL C01801 V=800.0 PL=0
MOVL C01802 V=800.0 PL=0
MOVL C01803 V=800.0 PL=0
MOVL C01804 V=800.0 PL=0
MOVL C01805 V=800.0 PL=0
MOVL C01806 V=800.0 PL=0
MOVL C01807 V=800.0 PL=0
MOVL C01808 V=800.0 PL=0
MOVL C01809 V=800.0 PL=0
MOVL C01810 V=800.0 PL=0
MOVL C01811 V=800.0 PL=0
MOVL C01812 V=800.0 PL=0
MOVL C01813 V=800.0 PL=0
MOVL C01814 V=800.0 PL=0
MOVL C01815 V=800.0 PL=0
MOVL C01816 V=800.0 PL=0
MOVL C01817 V=800.0 PL=0
MOVL C01818 V=800.0 PL=0
MOVL C01819 V=800.0 PL=0
MOVL C01820 V=800.0 PL=0
MOVL C01821 V=800.0 PL=0
MOVL C01822 V=800.0 PL=0
MOVL C01823 V=800.0 PL=0
MOVL C01824 V=800.0 PL=0
MOVL C01825 V=800.0 PL=0
MOVL C01826 V=800.0 PL=0
MOVL C01827 V=800.0 PL=0
MOVL C01828 V=800.0 PL=0
MOVL C01829 V=800.0 PL=0
MOVL C01830 V=800.0 PL=0
MOVL C01831 V=800.0 PL=0
MOVL C01832 V=800.0 PL=0
MOVL C01833 V=800.0 PL=0
MOVL C01834 V=800.0 PL=0
MOVL C01835 V=800.0 PL=0
MOVL C01836 V=800.0 PL=0
MOVL C01837 V=800.0 PL=0
MOVL C01838 V=800.0 PL=0
MOVL C01839 V=800.0 PL=0
MOVL C01840 V=800.0 PL=0
MOVL C01841 V=800.0 PL=0
MOVL C01842 V=800.0 PL=0
MOVL C01843 V=800.0 PL=0
MOVL C01844 V=800.0 PL=0
MOVL C01845 V=800.0 PL=0
MOVL C01846 V=800.0 PL=0
MOVL C01847 V=800.0 PL=0
MOVL C01848 V=800.0 PL=0
MOVL C01849 V=800.0 PL=0
MOVL C01850 V=800.0 PL=0
MOVL C01851 V=800.0 PL=0
MOVL C01852 V=800.0 PL=0
MOVL C01853 V=800.0 PL=0
MOVL C01854 V=800.0 PL=0
MOVL C01855 V=800.0 PL=0
MOVL C01856 V=800.0 PL=0
MOVL C01857 V=800.0 PL=0
MOVL C01858 V=800.0 PL=0
MOVL C01859 V=800.0 PL=0
MOVL C01860 V=800.0 PL=0
MOVL C01861 V=800.0 PL=0
MOVL C01862 V=800.0 PL=0
MOVL C01863 V=800.0 PL=0
MOVL C01864 V=800.0 PL=0
MOVL C01865 V=800.0 PL=0
MOVL C01866 V=800.0 PL=0
MOVL C01867 V=800.0 PL=0
MOVL C01868 V=800.0 PL=0
MOVL C01869 V=800.0 PL=0
MOVL C01870 V=800.0 PL=0
MOVL C01871 V=800.0 PL=0
MOVL C01872 V=800.0 PL=0
MOVL C01873 V=800.0 PL=0
MOVL C01874 V=800.0 PL=0
MOVL C01875 V=800.0 PL=0
MOVL C01876 V=800.0 PL=0
MOVL C01877 V=800.0 PL=0
MOVL C01878 V=800.0 PL=0
MOVL C01879 V=800.0 PL=0
MOVL C01880 V=800.0 PL=0
MOVL C01881 V=800.0 PL=0
MOVL C01882 V=800.0 PL=0
MOVL C01883 V=800.0 PL=0
MOVL C01884 V=800.0 PL=0
MOVL C01885 V=800.0 PL=0
MOVL C01886 V=800.0 PL=0
MOVL C01887 V=800.0 PL=0
MOVL C01888 V=800.0 PL=0
MOVL C01889 V=800.0 PL=0
MOVL C01890 V=800.0 PL=0
MOVL C01891 V=800.0 PL=0
MOVL C01892 V=800.0 PL=0
MOVL C01893 V=800.0 PL=0
MOVL C01894 V=800.0 PL=0
MOVL C01895 V=800.0 PL=0
MOVL C01896 V=800.0 PL=0
MOVL C01897 V=800.0 PL=0
MOVL C01898 V=800.0 PL=0
MOVL C01899 V=800.0 PL=0
MOVL C01900 V=800.0 PL=0
MOVL C01901 V=800.0 PL=0
MOVL C01902 V=800.0 PL=0
MOVL C01903 V=800.0 PL=0
MOVL C01904 V=800.0 PL=0
MOVL C01905 V=800.0 PL=0
MOVL C01906 V=800.0 PL=0
MOVL C01907 V=800.0 PL=0
MOVL C01908 V=800.0 PL=0
MOVL C01909 V=800.0 PL=0
MOVL C01910 V=800.0 PL=0
MOVL C01911 V=800.0 PL=0
MOVL C01912 V=800.0 PL=0
MOVL C01913 V=800.0 PL=0
MOVL C01914 V=800.0 PL=0
MOVL C01915 V=800.0 PL=0
MOVL C01916 V=800.0 PL=0
MOVL C01917 V=800.0 PL=0
MOVL C01918 V=800.0 PL=0
MOVL C01919 V=800.0 PL=0
MOVL C01920 V=800.0 PL=0
MOVL C01921 V=800.0 PL=0
MOVL C01922 V=800.0 PL=0
MOVL C01923 V=800.0 PL=0
MOVL C01924 V=800.0 PL=0
MOVL C01925 V=800.0 PL=0
MOVL C01926 V=800.0 PL=0
MOVL C01927 V=800.0 PL=0
MOVL C01928 V=800.0 PL=0
MOVL C01929 V=800.0 PL=0
MOVL C01930 V=800.0 PL=0
MOVL C01931 V=800.0 PL=0
MOVL C01932 V=800.0 PL=0
MOVL C01933 V=800.0 PL=0
MOVL C01934 V=800.0 PL=0
MOVL C01935 V=800.0 PL=0
MOVL C01936 V=800.0 PL=0
MOVL C01937 V=800.0 PL=0
MOVL C01938 V=800.0 PL=0
MOVL C01939 V=800.0 PL=0
MOVL C01940 V=800.0 PL=0
MOVL C01941 V=800.0 PL=0
MOVL C01942 V=800.0 PL=0
MOVL C01943 V=800.0 PL=0
MOVL C01944 V=800.0 PL=0
MOVL C01945 V=800.0 PL=0
MOVL C01946 V=800.0 PL=0
MOVL C01947 V=800.0 PL=0
MOVL C01948 V=800.0 PL=0
MOVL C01949 V=800.0 PL=0
MOVL C01950 V=800.0 PL=0
MOVL C01951 V=800.0 PL=0
MOVL C01952 V=800.0 PL=0
MOVL C01953 V=800.0 PL=0
MOVL C01954 V=800.0 PL=0
MOVL C01955 V=800.0 PL=0
MOVL C01956 V=800.0 PL=0
MOVL C01957 V=800.0 PL=0
MOVL C01958 V=800.0 PL=0
MOVL C01959 V=800.0 PL=0
MOVL C01960 V=800.0 PL=0
MOVL C01961 V=800.0 PL=0
MOVL C01962 V=800.0 PL=0
MOVL C01963 V=800.0 PL=0
MOVL C01964 V=800.0 PL=0
MOVL C01965 V=800.0 PL=0
MOVL C01966 V=800.0 PL=0
MOVL C01967 V=800.0 PL=0
MOVL C01968 V=800.0 PL=0
MOVL C01969 V=800.0 PL=0
MOVL C01970 V=800.0 PL=0
MOVL C01971 V=800.0 PL=0
MOVL C01972 V=800.0 PL=0
MOVL C01973 V=800.0 PL=0
MOVL C01974 V=800.0 PL=0
MOVL C01975 V=800.0 PL=0
MOVL C01976 V=800.0 PL=0
MOVL C01977 V=800.0 PL=0
MOVL C01978 V=800.0 PL=0
MOVL C01979 V=800.0 PL=0
MOVL C01980 V=800.0 PL=0
MOVL C01981 V=800.0 PL=0
MOVL C01982 V=800.0 PL=0
MOVL C01983 V=800.0 PL=0
MOVL C01984 V=800.0 PL=0
MOVL C01985 V=800.0 PL=0
MOVL C01986 V=800.0 PL=0
MOVL C01987 V=800.0 PL=0
MOVL C01988 V=800.0 PL=0
MOVL C01989 V=800.0 PL=0
MOVL C01990 V=800.0 PL=0
MOVL C01991 V=800.0 PL=0
MOVL C01992 V=800.0 PL=0
MOVL C01993 V=800.0 PL=0
MOVL C01994 V=800.0 PL=0
MOVL C01995 V=800.0 PL=0
MOVL C01996 V=800.0 PL=0
MOVL C01997 V=800.0 PL=0
MOVL C01998 V=800.0 PL=0
MOVL C01999 V=800.0 PL=0
MOVL C02000 V=800.0 PL=0
MOVL C02001 V=800.0 PL=0
MOVL C02002 V=800.0 PL=0
MOVL C02003 V=800.0 PL=0
MOVL C02004 V=800.0 PL=0
MOVL C02005 V=800.0 PL=0
MOVL C02006 V=800.0 PL=0
MOVL C02007 V=800.0 PL=0
MOVL C02008 V=800.0 PL=0
MOVL C02009 V=800.0 PL=0
MOVL C02010 V=800.0 PL=0
MOVL C02011 V=800.0 PL=0
MOVL C02012 V=800.0 PL=0
MOVL C02013 V=800.0 PL=0
MOVL C02014 V=800.0 PL=0
MOVL C02015 V=800.0 PL=0
MOVL C02016 V=800.0 PL=0
MOVL C02017 V=800.0 PL=0
MOVL C02018 V=800.0 PL=0
MOVL C02019 V=800.0 PL=0
MOVL C02020 V=800.0 PL=0
MOVL C02021 V=800.0 PL=0
MOVL C02022 V=800.0 PL=0
MOVL C02023 V=800.0 PL=0
MOVL C02024 V=800.0 PL=0
MOVL C02025 V=800.0 PL=0
MOVL C02026 V=800.0 PL=0
MOVL C02027 V=800.0 PL=0
MOVL C02028 V=800.0 PL=0
MOVL C02029 V=800.0 PL=0
MOVL C02030 V=800.0 PL=0
MOVL C02031 V=800.0 PL=0
MOVL C02032 V=800.0 PL=0
MOVL C02033 V=800.0 PL=0
MOVL C02034 V=800.0 PL=0
MOVL C02035 V=800.0 PL=0
MOVL C02036 V=800.0 PL=0
MOVL C02037 V=800.0 PL=0
MOVL C02038 V=800.0 PL=0
MOVL C02039 V=800.0 PL=0
MOVL C02040 V=800.0 PL=0
MOVL C02041 V=800.0 PL=0
MOVL C02042 V=800.0 PL=0
MOVL C02043 V=800.0 PL=0
MOVL C02044 V=800.0 PL=0
MOVL C02045 V=800.0 PL=0
MOVL C02046 V=800.0 PL=0
MOVL C02047 V=800.0 PL=0
MOVL C02048 V=800.0 PL=0
MOVL C02049 V=800.0 PL=0
MOVL C02050 V=800.0 PL=0
MOVL C02051 V=800.0 PL=0
MOVL C02052 V=800.0 PL=0
MOVL C02053 V=800.0 PL=0
MOVL C02054 V=800.0 PL=0
MOVL C02055 V=800.0 PL=0
MOVL C02056 V=800.0 PL=0
MOVL C02057 V=800.0 PL=0
MOVL C02058 V=800.0 PL=0
MOVL C02059 V=800.0 PL=0
MOVL C02060 V=800.0 PL=0
MOVL C02061 V=800.0 PL=0
MOVL C02062 V=800.0 PL=0
MOVL C02063 V=800.0 PL=0
MOVL C02064 V=800.0 PL=0
MOVL C02065 V=800.0 PL=0
MOVL C02066 V=800.0 PL=0
MOVL C02067 V=800.0 PL=0
MOVL C02068 V=800.0 PL=0
MOVL C02069 V=800.0 PL=0
MOVL C02070 V=800.0 PL=0
MOVL C02071 V=800.0 PL=0
MOVL C02072 V=800.0 PL=0
MOVL C02073 V=800.0 PL=0
MOVL C02074 V=800.0 PL=0
MOVL C02075 V=800.0 PL=0
MOVL C02076 V=800.0 PL=0
MOVL C02077 V=800.0 PL=0
MOVL C02078 V=800.0 PL=0
MOVL C02079 V=800.0 PL=0
MOVL C02080 V=800.0 PL=0
MOVL C02081 V=800.0 PL=0
MOVL C02082 V=800.0 PL=0
MOVL C02083 V=800.0 PL=0
MOVL C02084 V=800.0 PL=0
MOVL C02085 V=800.0 PL=0
MOVL C02086 V=800.0 PL=0
MOVL C02087 V=800.0 PL=0
MOVL C02088 V=800.0 PL=0
MOVL C02089 V=800.0 PL=0
MOVL C02090 V=800.0 PL=0
MOVL C02091 V=800.0 PL=0
MOVL C02092 V=800.0 PL=0
MOVL C02093 V=800.0 PL=0
MOVL C02094 V=800.0 PL=0
MOVL C02095 V=800.0 PL=0
MOVL C02096 V=800.0 PL=0
MOVL C02097 V=800.0 PL=0
MOVL C02098 V=800.0 PL=0
MOVL C02099 V=800.0 PL=0
MOVL C02100 V=800.0 PL=0
MOVL C02101 V=800.0 PL=0
MOVL C02102 V=800.0 PL=0
MOVL C02103 V=800.0 PL=0
MOVL C02104 V=800.0 PL=0
MOVL C02105 V=800.0 PL=0
MOVL C02106 V=800.0 PL=0
MOVL C02107 V=800.0 PL=0
MOVL C02108 V=800.0 PL=0
MOVL C02109 V=800.0 PL=0
MOVL C02110 V=800.0 PL=0
MOVL C02111 V=800.0 PL=0
MOVL C02112 V=800.0 PL=0
MOVL C02113 V=800.0 PL=0
MOVL C02114 V=800.0 PL=0
MOVL C02115 V=800.0 PL=0
MOVL C02116 V=800.0 PL=0
MOVL C02117 V=800.0 PL=0
MOVL C02118 V=800.0 PL=0
MOVL C02119 V=800.0 PL=0
MOVL C02120 V=800.0 PL=0
MOVL C02121 V=800.0 PL=0
MOVL C02122 V=800.0 PL=0
MOVL C02123 V=800.0 PL=0
MOVL C02124 V=800.0 PL=0
MOVL C02125 V=800.0 PL=0
MOVL C02126 V=800.0 PL=0
MOVL C02127 V=800.0 PL=0
MOVL C02128 V=800.0 PL=0
MOVL C02129 V=800.0 PL=0
MOVL C02130 V=800.0 PL=0
MOVL C02131 V=800.0 PL=0
MOVL C02132 V=800.0 PL=0
MOVL C02133 V=800.0 PL=0
MOVL C02134 V=800.0 PL=0
MOVL C02135 V=800.0 PL=0
MOVL C02136 V=800.0 PL=0
MOVL C02137 V=800.0 PL=0
MOVL C02138 V=800.0 PL=0
MOVL C02139 V=800.0 PL=0
MOVL C02140 V=800.0 PL=0
